Universal Robots PolyScope program: 2024.urp

Program 2024 (installation=default directory=/programs createdIn=5.11.9.1010452 lastSavedIn=5.11.9.1010452 robotSerialNumber=20225200364)
Calibrated DH parameters: a=[0.00002, -0.569483, -0.54992, -0.00001, -0.000036, 0]; d=[0.180894, -146.691669, 192.918669, -46.053088, 0.119778, 0.115602]; alpha=[1.571425, -0.001534, 0.003359, 1.568739, -1.571477, 0]; deltaTheta=[0, 0.376258, -0.101074, -0.275185, -0.000002, 0]
Robot Program (runOnlyOnce=true)
  Script file /programs/usbdisk/new-robot/2024Dragon_V2.script
    | def Machining1():
    |   # Default parameters:
    |   global speed_ms = 0.3
    |   global speed_rads = 0.75
    |   global accel_mss = 3
    |   global accel_radss = 1.2
    |   global blend_radius_m = 0.001
    | 
    |   # Add subprograms here
    |   # Start of main program
    |   # Program generated by RoboDK v5.6.5 for UR10e on 10/01/2024 16:52:19
    |   # Using nominal kinematics.
    |   blend_radius_m = 0.001
    |   speed_ms = 1.000
    |   # set_reference(p[0.320000, -0.152000, -0.016000, 0.000000, 0.000000, 0.000000])
    |   set_tcp(p[0.000000, 0.000000, 0.252000, 0.000000, 0.000000, 0.000000])
    |   # Show Tool
    |   movej([0.070455, -1.061149, -2.628944, -1.022296, 1.570796, 1.641252],accel_radss,speed_rads,0,blend_radius_m)
    |   movel([0.070455, -1.061149, -2.628944, -1.022296, 1.570796, 1.641252],accel_mss,speed_ms,0,blend_radius_m)
    |   # Splitting Linear movement in 30 (instruction 7: MoveL 3)
    |   movel([0.070455, -1.062891, -2.630322, -1.019175, 1.570796, 1.641252],accel_mss,speed_ms,0,blend_radius_m)
    |   movel([0.070455, -1.064646, -2.631698, -1.016044, 1.570796, 1.641252],accel_mss,speed_ms,0,blend_radius_m)
    |   movel([0.070455, -1.066415, -2.633072, -1.012903, 1.570796, 1.641252],accel_mss,speed_ms,0,blend_radius_m)
    |   movel([0.070455, -1.068196, -2.634443, -1.009750, 1.570796, 1.641252],accel_mss,speed_ms,0,blend_radius_m)
    |   movel([0.070455, -1.069991, -2.635811, -1.006586, 1.570796, 1.641252],accel_mss,speed_ms,0,blend_radius_m)
    |   movel([0.070455, -1.071800, -2.637177, -1.003412, 1.570796, 1.641252],accel_mss,speed_ms,0,blend_radius_m)
    |   movel([0.070455, -1.073622, -2.638541, -1.000227, 1.570796, 1.641252],accel_mss,speed_ms,0,blend_radius_m)
    |   movel([0.070455, -1.075457, -2.639902, -0.997030, 1.570796, 1.641252],accel_mss,speed_ms,0,blend_radius_m)
    |   movel([0.070455, -1.077307, -2.641260, -0.993822, 1.570796, 1.641252],accel_mss,speed_ms,0,blend_radius_m)
    |   movel([0.070455, -1.079170, -2.642616, -0.990603, 1.570796, 1.641252],accel_mss,speed_ms,0,blend_radius_m)
    |   movel([0.070455, -1.081047, -2.643969, -0.987373, 1.570796, 1.641252],accel_mss,speed_ms,0,blend_radius_m)
    |   movel([0.070455, -1.082937, -2.645320, -0.984132, 1.570796, 1.641252],accel_mss,speed_ms,0,blend_radius_m)
    |   movel([0.070455, -1.084842, -2.646667, -0.980879, 1.570796, 1.641252],accel_mss,speed_ms,0,blend_radius_m)
    |   movel([0.070455, -1.086761, -2.648013, -0.977615, 1.570796, 1.641252],accel_mss,speed_ms,0,blend_radius_m)
    |   movel([0.070455, -1.088694, -2.649355, -0.974339, 1.570796, 1.641252],accel_mss,speed_ms,0,blend_radius_m)
    |   movel([0.070455, -1.090642, -2.650695, -0.971052, 1.570796, 1.641252],accel_mss,speed_ms,0,blend_radius_m)
    |   movel([0.070455, -1.092603, -2.652032, -0.967753, 1.570796, 1.641252],accel_mss,speed_ms,0,blend_radius_m)
    |   movel([0.070455, -1.094579, -2.653367, -0.964443, 1.570796, 1.641252],accel_mss,speed_ms,0,blend_radius_m)
    |   movel([0.070455, -1.096570, -2.654698, -0.961121, 1.570796, 1.641252],accel_mss,speed_ms,0,blend_radius_m)
    |   movel([0.070455, -1.098575, -2.656027, -0.957787, 1.570796, 1.641252],accel_mss,speed_ms,0,blend_radius_m)
    |   movel([0.070455, -1.100594, -2.657353, -0.954441, 1.570796, 1.641252],accel_mss,speed_ms,0,blend_radius_m)
    |   movel([0.070455, -1.102629, -2.658677, -0.951083, 1.570796, 1.641252],accel_mss,speed_ms,0,blend_radius_m)
    |   movel([0.070455, -1.104678, -2.659997, -0.947714, 1.570796, 1.641252],accel_mss,speed_ms,0,blend_radius_m)
    |   movel([0.070455, -1.106742, -2.661315, -0.944332, 1.570796, 1.641252],accel_mss,speed_ms,0,blend_radius_m)
    |   movel([0.070455, -1.108821, -2.662630, -0.940938, 1.570796, 1.641252],accel_mss,speed_ms,0,blend_radius_m)
    |   movel([0.070455, -1.110915, -2.663942, -0.937533, 1.570796, 1.641252],accel_mss,speed_ms,0,blend_radius_m)
    |   movel([0.070455, -1.113024, -2.665251, -0.934115, 1.570796, 1.641252],accel_mss,speed_ms,0,blend_radius_m)
    |   movel([0.070455, -1.115148, -2.666557, -0.930684, 1.570796, 1.641252],accel_mss,speed_ms,0,blend_radius_m)
    |   movel([0.070455, -1.117287, -2.667860, -0.927242, 1.570796, 1.641252],accel_mss,speed_ms,0,blend_radius_m)
    |   movel([0.070455, -1.119442, -2.669160, -0.923787, 1.570796, 1.641252],accel_mss,speed_ms,0,blend_radius_m)
    |   movel([0.070455, -1.119442, -2.669160, -0.923787, 1.570796, 1.641252],accel_mss,speed_ms,0,blend_radius_m)
    |   speed_ms = 1.000
    |   movel([0.070455, -1.119442, -2.669160, -0.923787, 1.570796, 1.641252],accel_mss,speed_ms,0,blend_radius_m)
    |   movel([0.070455, -1.119442, -2.669160, -0.923787, 1.570796, 1.641252],accel_mss,speed_ms,0,blend_radius_m)
    |   movel([0.070455, -1.119442, -2.669160, -0.923787, 1.570796, 1.641252],accel_mss,speed_ms,0,blend_radius_m)
    |   speed_ms = 0.005
    |   # Splitting Linear movement in 20 (instruction 14: MoveL 8)
    |   movel([0.070455, -1.117287, -2.667860, -0.927242, 1.570796, 1.641252],accel_mss,speed_ms,0,blend_radius_m)
    |   movel([0.070455, -1.115148, -2.666557, -0.930684, 1.570796, 1.641252],accel_mss,speed_ms,0,blend_radius_m)
    |   movel([0.070455, -1.113024, -2.665251, -0.934115, 1.570796, 1.641252],accel_mss,speed_ms,0,blend_radius_m)
    |   movel([0.070455, -1.110915, -2.663942, -0.937533, 1.570796, 1.641252],accel_mss,speed_ms,0,blend_radius_m)
    |   movel([0.070455, -1.108821, -2.662630, -0.940938, 1.570796, 1.641252],accel_mss,speed_ms,0,blend_radius_m)
    |   movel([0.070455, -1.106742, -2.661315, -0.944332, 1.570796, 1.641252],accel_mss,speed_ms,0,blend_radius_m)
    |   movel([0.070455, -1.104678, -2.659997, -0.947714, 1.570796, 1.641252],accel_mss,speed_ms,0,blend_radius_m)
    |   movel([0.070455, -1.102629, -2.658677, -0.951083, 1.570796, 1.641252],accel_mss,speed_ms,0,blend_radius_m)
    |   movel([0.070455, -1.100594, -2.657353, -0.954441, 1.570796, 1.641252],accel_mss,speed_ms,0,blend_radius_m)
    |   movel([0.070455, -1.098575, -2.656027, -0.957787, 1.570796, 1.641252],accel_mss,speed_ms,0,blend_radius_m)
    |   movel([0.070455, -1.096570, -2.654698, -0.961121, 1.570796, 1.641252],accel_mss,speed_ms,0,blend_radius_m)
    |   movel([0.070455, -1.094579, -2.653367, -0.964443, 1.570796, 1.641252],accel_mss,speed_ms,0,blend_radius_m)
    |   movel([0.070455, -1.092603, -2.652032, -0.967753, 1.570796, 1.641252],accel_mss,speed_ms,0,blend_radius_m)
    |   movel([0.070455, -1.090642, -2.650695, -0.971052, 1.570796, 1.641252],accel_mss,speed_ms,0,blend_radius_m)
    |   movel([0.070455, -1.088694, -2.649355, -0.974339, 1.570796, 1.641252],accel_mss,speed_ms,0,blend_radius_m)
    |   movel([0.070455, -1.086761, -2.648013, -0.977615, 1.570796, 1.641252],accel_mss,speed_ms,0,blend_radius_m)
    |   movel([0.070455, -1.084842, -2.646667, -0.980879, 1.570796, 1.641252],accel_mss,speed_ms,0,blend_radius_m)
    |   movel([0.070455, -1.082937, -2.645320, -0.984132, 1.570796, 1.641252],accel_mss,speed_ms,0,blend_radius_m)
    |   movel([0.070455, -1.081047, -2.643969, -0.987373, 1.570796, 1.641252],accel_mss,speed_ms,0,blend_radius_m)
    |   movel([0.070455, -1.079170, -2.642616, -0.990603, 1.570796, 1.641252],accel_mss,speed_ms,0,blend_radius_m)
    |   speed_ms = 1.000
    |   # Splitting Linear movement in 20 (instruction 16: MoveL 9)
    |   movel([0.070455, -1.081047, -2.643969, -0.987373, 1.570796, 1.641252],accel_mss,speed_ms,0,blend_radius_m)
    |   movel([0.070455, -1.082937, -2.645320, -0.984132, 1.570796, 1.641252],accel_mss,speed_ms,0,blend_radius_m)
    |   movel([0.070455, -1.084842, -2.646667, -0.980879, 1.570796, 1.641252],accel_mss,speed_ms,0,blend_radius_m)
    |   movel([0.070455, -1.086761, -2.648013, -0.977615, 1.570796, 1.641252],accel_mss,speed_ms,0,blend_radius_m)
    |   movel([0.070455, -1.088694, -2.649355, -0.974339, 1.570796, 1.641252],accel_mss,speed_ms,0,blend_radius_m)
    |   movel([0.070455, -1.090642, -2.650695, -0.971052, 1.570796, 1.641252],accel_mss,speed_ms,0,blend_radius_m)
    |   movel([0.070455, -1.092603, -2.652032, -0.967753, 1.570796, 1.641252],accel_mss,speed_ms,0,blend_radius_m)
    |   movel([0.070455, -1.094579, -2.653367, -0.964443, 1.570796, 1.641252],accel_mss,speed_ms,0,blend_radius_m)
    |   movel([0.070455, -1.096570, -2.654698, -0.961121, 1.570796, 1.641252],accel_mss,speed_ms,0,blend_radius_m)
    |   movel([0.070455, -1.098575, -2.656027, -0.957787, 1.570796, 1.641252],accel_mss,speed_ms,0,blend_radius_m)
    |   movel([0.070455, -1.100594, -2.657353, -0.954441, 1.570796, 1.641252],accel_mss,speed_ms,0,blend_radius_m)
    |   movel([0.070455, -1.102629, -2.658677, -0.951083, 1.570796, 1.641252],accel_mss,speed_ms,0,blend_radius_m)
    |   movel([0.070455, -1.104678, -2.659997, -0.947714, 1.570796, 1.641252],accel_mss,speed_ms,0,blend_radius_m)
    |   movel([0.070455, -1.106742, -2.661315, -0.944332, 1.570796, 1.641252],accel_mss,speed_ms,0,blend_radius_m)
    |   movel([0.070455, -1.108821, -2.662630, -0.940938, 1.570796, 1.641252],accel_mss,speed_ms,0,blend_radius_m)
    |   movel([0.070455, -1.110915, -2.663942, -0.937533, 1.570796, 1.641252],accel_mss,speed_ms,0,blend_radius_m)
    |   movel([0.070455, -1.113024, -2.665251, -0.934115, 1.570796, 1.641252],accel_mss,speed_ms,0,blend_radius_m)
    |   movel([0.070455, -1.115148, -2.666557, -0.930684, 1.570796, 1.641252],accel_mss,speed_ms,0,blend_radius_m)
    |   movel([0.070455, -1.117287, -2.667860, -0.927242, 1.570796, 1.641252],accel_mss,speed_ms,0,blend_radius_m)
    |   movel([0.070455, -1.119442, -2.669160, -0.923787, 1.570796, 1.641252],accel_mss,speed_ms,0,blend_radius_m)
    |   speed_ms = 0.040
    |   movel([0.070455, -1.119442, -2.669160, -0.923787, 1.570796, 1.641252],accel_mss,speed_ms,0,blend_radius_m)
    |   speed_ms = 1.000
    |   movel([0.070455, -1.119442, -2.669160, -0.923787, 1.570796, 1.641252],accel_mss,speed_ms,0,blend_radius_m)
    |   # Splitting Linear movement in 152 (instruction 21: MoveL 12)
    |   movel([0.070832, -1.122077, -2.668067, -0.922246, 1.570796, 1.641628],accel_mss,speed_ms,0,blend_radius_m)
    |   movel([0.071206, -1.124704, -2.666969, -0.920715, 1.570796, 1.642002],accel_mss,speed_ms,0,blend_radius_m)
    |   movel([0.071578, -1.127324, -2.665869, -0.919196, 1.570796, 1.642374],accel_mss,speed_ms,0,blend_radius_m)
    |   movel([0.071947, -1.129937, -2.664764, -0.917688, 1.570796, 1.642743],accel_mss,speed_ms,0,blend_radius_m)
    |   movel([0.072314, -1.132542, -2.663657, -0.916190, 1.570796, 1.643111],accel_mss,speed_ms,0,blend_radius_m)
    |   movel([0.072679, -1.135140, -2.662545, -0.914703, 1.570796, 1.643476],accel_mss,speed_ms,0,blend_radius_m)
    |   movel([0.073042, -1.137731, -2.661431, -0.913227, 1.570796, 1.643839],accel_mss,speed_ms,0,blend_radius_m)
    |   movel([0.073403, -1.140315, -2.660313, -0.911762, 1.570796, 1.644199],accel_mss,speed_ms,0,blend_radius_m)
    |   movel([0.073761, -1.142891, -2.659192, -0.910307, 1.570796, 1.644558],accel_mss,speed_ms,0,blend_radius_m)
    |   movel([0.074117, -1.145460, -2.658067, -0.908863, 1.570796, 1.644914],accel_mss,speed_ms,0,blend_radius_m)
    |   movel([0.074472, -1.148021, -2.656939, -0.907429, 1.570796, 1.645268],accel_mss,speed_ms,0,blend_radius_m)
    |   movel([0.074824, -1.150576, -2.655807, -0.906006, 1.570796, 1.645620],accel_mss,speed_ms,0,blend_radius_m)
    |   movel([0.075173, -1.153123, -2.654672, -0.904594, 1.570796, 1.645970],accel_mss,speed_ms,0,blend_radius_m)
    |   movel([0.075521, -1.155663, -2.653534, -0.903192, 1.570796, 1.646318],accel_mss,speed_ms,0,blend_radius_m)
    |   movel([0.075867, -1.158196, -2.652393, -0.901800, 1.570796, 1.646663],accel_mss,speed_ms,0,blend_radius_m)
    |   movel([0.076211, -1.160722, -2.651248, -0.900419, 1.570796, 1.647007],accel_mss,speed_ms,0,blend_radius_m)
    |   movel([0.076552, -1.163240, -2.650100, -0.899048, 1.570796, 1.647349],accel_mss,speed_ms,0,blend_radius_m)
    |   movel([0.076892, -1.165752, -2.648949, -0.897688, 1.570796, 1.647688],accel_mss,speed_ms,0,blend_radius_m)
    |   movel([0.077230, -1.168256, -2.647795, -0.896338, 1.570796, 1.648026],accel_mss,speed_ms,0,blend_radius_m)
    |   movel([0.077565, -1.170754, -2.646637, -0.894998, 1.570796, 1.648362],accel_mss,speed_ms,0,blend_radius_m)
    |   movel([0.077899, -1.173244, -2.645477, -0.893668, 1.570796, 1.648695],accel_mss,speed_ms,0,blend_radius_m)
    |   movel([0.078231, -1.175728, -2.644313, -0.892348, 1.570796, 1.649027],accel_mss,speed_ms,0,blend_radius_m)
    |   movel([0.078561, -1.178204, -2.643146, -0.891039, 1.570796, 1.649357],accel_mss,speed_ms,0,blend_radius_m)
    |   movel([0.078888, -1.180674, -2.641976, -0.889739, 1.570796, 1.649685],accel_mss,speed_ms,0,blend_radius_m)
    |   movel([0.079214, -1.183137, -2.640802, -0.888450, 1.570796, 1.650011],accel_mss,speed_ms,0,blend_radius_m)
    |   movel([0.079539, -1.185593, -2.639626, -0.887171, 1.570796, 1.650335],accel_mss,speed_ms,0,blend_radius_m)
    |   movel([0.079861, -1.188042, -2.638446, -0.885901, 1.570796, 1.650657],accel_mss,speed_ms,0,blend_radius_m)
    |   movel([0.080181, -1.190484, -2.637264, -0.884642, 1.570796, 1.650978],accel_mss,speed_ms,0,blend_radius_m)
    |   movel([0.080500, -1.192919, -2.636078, -0.883392, 1.570796, 1.651296],accel_mss,speed_ms,0,blend_radius_m)
    |   movel([0.080817, -1.195347, -2.634889, -0.882152, 1.570796, 1.651613],accel_mss,speed_ms,0,blend_radius_m)
    |   movel([0.081131, -1.197769, -2.633698, -0.880922, 1.570796, 1.651928],accel_mss,speed_ms,0,blend_radius_m)
    |   movel([0.081445, -1.200184, -2.632503, -0.879702, 1.570796, 1.652241],accel_mss,speed_ms,0,blend_radius_m)
    |   movel([0.081756, -1.202593, -2.631305, -0.878491, 1.570796, 1.652552],accel_mss,speed_ms,0,blend_radius_m)
    |   movel([0.082066, -1.204994, -2.630105, -0.877290, 1.570796, 1.652862],accel_mss,speed_ms,0,blend_radius_m)
    |   movel([0.082374, -1.207389, -2.628901, -0.876099, 1.570796, 1.653170],accel_mss,speed_ms,0,blend_radius_m)
    |   movel([0.082680, -1.209777, -2.627694, -0.874917, 1.570796, 1.653476],accel_mss,speed_ms,0,blend_radius_m)
    |   movel([0.082984, -1.212159, -2.626485, -0.873745, 1.570796, 1.653780],accel_mss,speed_ms,0,blend_radius_m)
    |   movel([0.083287, -1.214534, -2.625272, -0.872582, 1.570796, 1.654083],accel_mss,speed_ms,0,blend_radius_m)
    |   movel([0.083588, -1.216903, -2.624057, -0.871429, 1.570796, 1.654384],accel_mss,speed_ms,0,blend_radius_m)
    |   movel([0.083887, -1.219265, -2.622839, -0.870285, 1.570796, 1.654684],accel_mss,speed_ms,0,blend_radius_m)
    |   movel([0.084185, -1.221621, -2.621618, -0.869151, 1.570796, 1.654981],accel_mss,speed_ms,0,blend_radius_m)
    |   movel([0.084481, -1.223970, -2.620394, -0.868026, 1.570796, 1.655277],accel_mss,speed_ms,0,blend_radius_m)
    |   movel([0.084775, -1.226312, -2.619167, -0.866910, 1.570796, 1.655572],accel_mss,speed_ms,0,blend_radius_m)
    |   movel([0.085068, -1.228649, -2.617937, -0.865803, 1.570796, 1.655864],accel_mss,speed_ms,0,blend_radius_m)
    |   movel([0.085359, -1.230978, -2.616705, -0.864706, 1.570796, 1.656156],accel_mss,speed_ms,0,blend_radius_m)
    |   movel([0.085649, -1.233302, -2.615469, -0.863618, 1.570796, 1.656445],accel_mss,speed_ms,0,blend_radius_m)
    |   movel([0.085937, -1.235619, -2.614231, -0.862539, 1.570796, 1.656733],accel_mss,speed_ms,0,blend_radius_m)
    |   movel([0.086223, -1.237930, -2.612991, -0.861468, 1.570796, 1.657020],accel_mss,speed_ms,0,blend_radius_m)
    |   movel([0.086508, -1.240234, -2.611747, -0.860407, 1.570796, 1.657304],accel_mss,speed_ms,0,blend_radius_m)
    |   movel([0.086791, -1.242533, -2.610501, -0.859355, 1.570796, 1.657588],accel_mss,speed_ms,0,blend_radius_m)
    |   movel([0.087073, -1.244825, -2.609252, -0.858312, 1.570796, 1.657869],accel_mss,speed_ms,0,blend_radius_m)
    |   movel([0.087353, -1.247111, -2.608000, -0.857278, 1.570796, 1.658150],accel_mss,speed_ms,0,blend_radius_m)
    |   movel([0.087632, -1.249390, -2.606746, -0.856253, 1.570796, 1.658428],accel_mss,speed_ms,0,blend_radius_m)
    |   movel([0.087909, -1.251664, -2.605488, -0.855237, 1.570796, 1.658706],accel_mss,speed_ms,0,blend_radius_m)
    |   movel([0.088185, -1.253931, -2.604229, -0.854229, 1.570796, 1.658981],accel_mss,speed_ms,0,blend_radius_m)
    |   movel([0.088459, -1.256193, -2.602966, -0.853230, 1.570796, 1.659256],accel_mss,speed_ms,0,blend_radius_m)
    |   movel([0.088732, -1.258448, -2.601701, -0.852240, 1.570796, 1.659528],accel_mss,speed_ms,0,blend_radius_m)
    |   movel([0.089004, -1.260697, -2.600433, -0.851258, 1.570796, 1.659800],accel_mss,speed_ms,0,blend_radius_m)
    |   movel([0.089273, -1.262941, -2.599163, -0.850285, 1.570796, 1.660070],accel_mss,speed_ms,0,blend_radius_m)
    |   movel([0.089542, -1.265178, -2.597890, -0.849321, 1.570796, 1.660338],accel_mss,speed_ms,0,blend_radius_m)
    |   movel([0.089809, -1.267409, -2.596614, -0.848365, 1.570796, 1.660605],accel_mss,speed_ms,0,blend_radius_m)
    |   movel([0.090075, -1.269635, -2.595336, -0.847418, 1.570796, 1.660871],accel_mss,speed_ms,0,blend_radius_m)
    |   movel([0.090339, -1.271854, -2.594055, -0.846479, 1.570796, 1.661135],accel_mss,speed_ms,0,blend_radius_m)
    |   movel([0.090602, -1.274068, -2.592772, -0.845549, 1.570796, 1.661398],accel_mss,speed_ms,0,blend_radius_m)
    |   movel([0.090863, -1.276276, -2.591486, -0.844627, 1.570796, 1.661660],accel_mss,speed_ms,0,blend_radius_m)
    |   movel([0.091123, -1.278478, -2.590198, -0.843713, 1.570796, 1.661920],accel_mss,speed_ms,0,blend_radius_m)
    |   movel([0.091382, -1.280674, -2.588907, -0.842808, 1.570796, 1.662178],accel_mss,speed_ms,0,blend_radius_m)
    |   movel([0.091640, -1.282864, -2.587614, -0.841911, 1.570796, 1.662436],accel_mss,speed_ms,0,blend_radius_m)
    |   movel([0.091896, -1.285049, -2.586318, -0.841022, 1.570796, 1.662692],accel_mss,speed_ms,0,blend_radius_m)
    |   movel([0.092150, -1.287228, -2.585019, -0.840141, 1.570796, 1.662947],accel_mss,speed_ms,0,blend_radius_m)
    |   movel([0.092404, -1.289402, -2.583719, -0.839269, 1.570796, 1.663200],accel_mss,speed_ms,0,blend_radius_m)
    |   movel([0.092656, -1.291569, -2.582415, -0.838404, 1.570796, 1.663452],accel_mss,speed_ms,0,blend_radius_m)
    |   movel([0.092907, -1.293731, -2.581110, -0.837548, 1.570796, 1.663703],accel_mss,speed_ms,0,blend_radius_m)
    |   movel([0.093156, -1.295888, -2.579801, -0.836700, 1.570796, 1.663953],accel_mss,speed_ms,0,blend_radius_m)
    |   movel([0.093405, -1.298039, -2.578491, -0.835859, 1.570796, 1.664201],accel_mss,speed_ms,0,blend_radius_m)
    |   movel([0.093652, -1.300184, -2.577178, -0.835027, 1.570796, 1.664448],accel_mss,speed_ms,0,blend_radius_m)
    |   movel([0.093897, -1.302324, -2.575862, -0.834202, 1.570796, 1.664694],accel_mss,speed_ms,0,blend_radius_m)
    |   movel([0.094142, -1.304459, -2.574545, -0.833386, 1.570796, 1.664938],accel_mss,speed_ms,0,blend_radius_m)
    |   movel([0.094385, -1.306588, -2.573224, -0.832577, 1.570796, 1.665182],accel_mss,speed_ms,0,blend_radius_m)
    |   movel([0.094627, -1.308711, -2.571902, -0.831776, 1.570796, 1.665424],accel_mss,speed_ms,0,blend_radius_m)
    |   movel([0.094868, -1.310829, -2.570577, -0.830983, 1.570796, 1.665664],accel_mss,speed_ms,0,blend_radius_m)
    |   movel([0.095108, -1.312942, -2.569250, -0.830197, 1.570796, 1.665904],accel_mss,speed_ms,0,blend_radius_m)
    |   movel([0.095346, -1.315050, -2.567920, -0.829419, 1.570796, 1.666142],accel_mss,speed_ms,0,blend_radius_m)
    |   movel([0.095583, -1.317152, -2.566588, -0.828649, 1.570796, 1.666380],accel_mss,speed_ms,0,blend_radius_m)
    |   movel([0.095819, -1.319249, -2.565254, -0.827886, 1.570796, 1.666616],accel_mss,speed_ms,0,blend_radius_m)
    |   movel([0.096054, -1.321340, -2.563918, -0.827131, 1.570796, 1.666851],accel_mss,speed_ms,0,blend_radius_m)
    |   movel([0.096288, -1.323427, -2.562579, -0.826384, 1.570796, 1.667084],accel_mss,speed_ms,0,blend_radius_m)
    |   movel([0.096520, -1.325508, -2.561238, -0.825643, 1.570796, 1.667317],accel_mss,speed_ms,0,blend_radius_m)
    |   movel([0.096752, -1.327584, -2.559894, -0.824911, 1.570796, 1.667548],accel_mss,speed_ms,0,blend_radius_m)
    |   movel([0.096982, -1.329654, -2.558549, -0.824186, 1.570796, 1.667778],accel_mss,speed_ms,0,blend_radius_m)
    |   movel([0.097211, -1.331720, -2.557201, -0.823468, 1.570796, 1.668007],accel_mss,speed_ms,0,blend_radius_m)
    |   movel([0.097439, -1.333781, -2.555851, -0.822757, 1.570796, 1.668235],accel_mss,speed_ms,0,blend_radius_m)
    |   movel([0.097666, -1.335836, -2.554499, -0.822054, 1.570796, 1.668462],accel_mss,speed_ms,0,blend_radius_m)
    |   movel([0.097892, -1.337887, -2.553144, -0.821358, 1.570796, 1.668688],accel_mss,speed_ms,0,blend_radius_m)
    |   movel([0.098116, -1.339932, -2.551787, -0.820669, 1.570796, 1.668913],accel_mss,speed_ms,0,blend_radius_m)
    |   movel([0.098340, -1.341972, -2.550429, -0.819988, 1.570796, 1.669136],accel_mss,speed_ms,0,blend_radius_m)
    |   movel([0.098562, -1.344008, -2.549067, -0.819314, 1.570796, 1.669359],accel_mss,speed_ms,0,blend_radius_m)
    |   movel([0.098784, -1.346038, -2.547704, -0.818646, 1.570796, 1.669580],accel_mss,speed_ms,0,blend_radius_m)
    |   movel([0.099004, -1.348064, -2.546339, -0.817986, 1.570796, 1.669800],accel_mss,speed_ms,0,blend_radius_m)
    |   movel([0.099223, -1.350085, -2.544971, -0.817333, 1.570796, 1.670020],accel_mss,speed_ms,0,blend_radius_m)
    |   movel([0.099441, -1.352100, -2.543601, -0.816687, 1.570796, 1.670238],accel_mss,speed_ms,0,blend_radius_m)
    |   movel([0.099659, -1.354111, -2.542230, -0.816048, 1.570796, 1.670455],accel_mss,speed_ms,0,blend_radius_m)
    |   movel([0.099875, -1.356118, -2.540856, -0.815416, 1.570796, 1.670671],accel_mss,speed_ms,0,blend_radius_m)
    |   movel([0.100090, -1.358119, -2.539479, -0.814791, 1.570796, 1.670886],accel_mss,speed_ms,0,blend_radius_m)
    |   movel([0.100304, -1.360116, -2.538101, -0.814172, 1.570796, 1.671100],accel_mss,speed_ms,0,blend_radius_m)
    |   movel([0.100517, -1.362107, -2.536721, -0.813561, 1.570796, 1.671313],accel_mss,speed_ms,0,blend_radius_m)
    |   movel([0.100729, -1.364095, -2.535338, -0.812956, 1.570796, 1.671525],accel_mss,speed_ms,0,blend_radius_m)
    |   movel([0.100940, -1.366077, -2.533954, -0.812358, 1.570796, 1.671736],accel_mss,speed_ms,0,blend_radius_m)
    |   movel([0.101150, -1.368055, -2.532567, -0.811767, 1.570796, 1.671946],accel_mss,speed_ms,0,blend_radius_m)
    |   movel([0.101359, -1.370028, -2.531179, -0.811182, 1.570796, 1.672155],accel_mss,speed_ms,0,blend_radius_m)
    |   movel([0.101567, -1.371997, -2.529788, -0.810604, 1.570796, 1.672363],accel_mss,speed_ms,0,blend_radius_m)
    |   movel([0.101774, -1.373961, -2.528395, -0.810033, 1.570796, 1.672570],accel_mss,speed_ms,0,blend_radius_m)
    |   movel([0.101980, -1.375920, -2.527000, -0.809468, 1.570796, 1.672776],accel_mss,speed_ms,0,blend_radius_m)
    |   movel([0.102185, -1.377875, -2.525604, -0.808910, 1.570796, 1.672981],accel_mss,speed_ms,0,blend_radius_m)
    |   movel([0.102389, -1.379825, -2.524205, -0.808359, 1.570796, 1.673186],accel_mss,speed_ms,0,blend_radius_m)
    |   movel([0.102593, -1.381771, -2.522804, -0.807814, 1.570796, 1.673389],accel_mss,speed_ms,0,blend_radius_m)
    |   movel([0.102795, -1.383713, -2.521401, -0.807275, 1.570796, 1.673591],accel_mss,speed_ms,0,blend_radius_m)
    |   movel([0.102996, -1.385650, -2.519996, -0.806743, 1.570796, 1.673792],accel_mss,speed_ms,0,blend_radius_m)
    |   movel([0.103197, -1.387582, -2.518589, -0.806217, 1.570796, 1.673993],accel_mss,speed_ms,0,blend_radius_m)
    |   movel([0.103396, -1.389510, -2.517181, -0.805698, 1.570796, 1.674192],accel_mss,speed_ms,0,blend_radius_m)
    |   movel([0.103595, -1.391434, -2.515770, -0.805185, 1.570796, 1.674391],accel_mss,speed_ms,0,blend_radius_m)
    |   movel([0.103792, -1.393354, -2.514357, -0.804678, 1.570796, 1.674588],accel_mss,speed_ms,0,blend_radius_m)
    |   movel([0.103989, -1.395269, -2.512942, -0.804178, 1.570796, 1.674785],accel_mss,speed_ms,0,blend_radius_m)
    |   movel([0.104185, -1.397180, -2.511526, -0.803684, 1.570796, 1.674981],accel_mss,speed_ms,0,blend_radius_m)
    |   movel([0.104380, -1.399086, -2.510107, -0.803196, 1.570796, 1.675176],accel_mss,speed_ms,0,blend_radius_m)
    |   movel([0.104574, -1.400989, -2.508686, -0.802714, 1.570796, 1.675370],accel_mss,speed_ms,0,blend_radius_m)
    |   movel([0.104767, -1.402887, -2.507264, -0.802238, 1.570796, 1.675563],accel_mss,speed_ms,0,blend_radius_m)
    |   movel([0.104959, -1.404781, -2.505840, -0.801769, 1.570796, 1.675755],accel_mss,speed_ms,0,blend_radius_m)
    |   movel([0.105151, -1.406670, -2.504413, -0.801305, 1.570796, 1.675947],accel_mss,speed_ms,0,blend_radius_m)
    |   movel([0.105341, -1.408556, -2.502985, -0.800848, 1.570796, 1.676137],accel_mss,speed_ms,0,blend_radius_m)
    |   movel([0.105531, -1.410437, -2.501555, -0.800397, 1.570796, 1.676327],accel_mss,speed_ms,0,blend_radius_m)
    |   movel([0.105720, -1.412315, -2.500123, -0.799951, 1.570796, 1.676516],accel_mss,speed_ms,0,blend_radius_m)
    |   movel([0.105908, -1.414188, -2.498689, -0.799512, 1.570796, 1.676704],accel_mss,speed_ms,0,blend_radius_m)
    |   movel([0.106095, -1.416057, -2.497254, -0.799078, 1.570796, 1.676891],accel_mss,speed_ms,0,blend_radius_m)
    |   movel([0.106281, -1.417922, -2.495816, -0.798651, 1.570796, 1.677077],accel_mss,speed_ms,0,blend_radius_m)
    |   movel([0.106466, -1.419783, -2.494377, -0.798229, 1.570796, 1.677263],accel_mss,speed_ms,0,blend_radius_m)
    |   movel([0.106651, -1.421640, -2.492935, -0.797813, 1.570796, 1.677447],accel_mss,speed_ms,0,blend_radius_m)
    |   movel([0.106835, -1.423494, -2.491492, -0.797403, 1.570796, 1.677631],accel_mss,speed_ms,0,blend_radius_m)
    |   movel([0.107018, -1.425343, -2.490047, -0.796999, 1.570796, 1.677814],accel_mss,speed_ms,0,blend_radius_m)
    |   movel([0.107200, -1.427188, -2.488600, -0.796600, 1.570796, 1.677997],accel_mss,speed_ms,0,blend_radius_m)
    |   movel([0.107382, -1.429030, -2.487152, -0.796208, 1.570796, 1.678178],accel_mss,speed_ms,0,blend_radius_m)
    |   movel([0.107562, -1.430867, -2.485701, -0.795821, 1.570796, 1.678359],accel_mss,speed_ms,0,blend_radius_m)
    |   movel([0.107742, -1.432701, -2.484249, -0.795439, 1.570796, 1.678538],accel_mss,speed_ms,0,blend_radius_m)
    |   movel([0.107921, -1.434531, -2.482795, -0.795063, 1.570796, 1.678717],accel_mss,speed_ms,0,blend_radius_m)
    |   movel([0.108099, -1.436357, -2.481339, -0.794693, 1.570796, 1.678896],accel_mss,speed_ms,0,blend_radius_m)
    |   movel([0.108277, -1.438179, -2.479881, -0.794329, 1.570796, 1.679073],accel_mss,speed_ms,0,blend_radius_m)
    |   movel([0.108453, -1.439997, -2.478422, -0.793970, 1.570796, 1.679250],accel_mss,speed_ms,0,blend_radius_m)
    |   movel([0.108629, -1.441812, -2.476961, -0.793616, 1.570796, 1.679426],accel_mss,speed_ms,0,blend_radius_m)
    |   movel([0.108804, -1.443623, -2.475498, -0.793268, 1.570796, 1.679601],accel_mss,speed_ms,0,blend_radius_m)
    |   movel([0.108979, -1.445430, -2.474033, -0.792926, 1.570796, 1.679775],accel_mss,speed_ms,0,blend_radius_m)
    |   movel([0.109152, -1.447233, -2.472567, -0.792589, 1.570796, 1.679949],accel_mss,speed_ms,0,blend_radius_m)
    |   movel([0.109325, -1.449033, -2.471098, -0.792257, 1.570796, 1.680122],accel_mss,speed_ms,0,blend_radius_m)
    |   speed_ms = 0.005
    |   # Splitting Linear movement in 20 (instruction 23: MoveL 13)
    |   movel([0.109325, -1.450882, -2.472048, -0.789459, 1.570796, 1.680122],accel_mss,speed_ms,0,blend_radius_m)
    |   movel([0.109325, -1.452738, -2.472994, -0.786657, 1.570796, 1.680122],accel_mss,speed_ms,0,blend_radius_m)
    |   movel([0.109325, -1.454601, -2.473936, -0.783852, 1.570796, 1.680122],accel_mss,speed_ms,0,blend_radius_m)
    |   movel([0.109325, -1.456472, -2.474875, -0.781042, 1.570796, 1.680122],accel_mss,speed_ms,0,blend_radius_m)
    |   movel([0.109325, -1.458351, -2.475811, -0.778228, 1.570796, 1.680122],accel_mss,speed_ms,0,blend_radius_m)
    |   movel([0.109325, -1.460236, -2.476742, -0.775410, 1.570796, 1.680122],accel_mss,speed_ms,0,blend_radius_m)
    |   movel([0.109325, -1.462130, -2.477671, -0.772588, 1.570796, 1.680122],accel_mss,speed_ms,0,blend_radius_m)
    |   movel([0.109325, -1.464030, -2.478596, -0.769763, 1.570796, 1.680122],accel_mss,speed_ms,0,blend_radius_m)
    |   movel([0.109325, -1.465939, -2.479517, -0.766933, 1.570796, 1.680122],accel_mss,speed_ms,0,blend_radius_m)
    |   movel([0.109325, -1.467854, -2.480435, -0.764100, 1.570796, 1.680122],accel_mss,speed_ms,0,blend_radius_m)
    |   movel([0.109325, -1.469778, -2.481349, -0.761262, 1.570796, 1.680122],accel_mss,speed_ms,0,blend_radius_m)
    |   movel([0.109325, -1.471708, -2.482260, -0.758421, 1.570796, 1.680122],accel_mss,speed_ms,0,blend_radius_m)
    |   movel([0.109325, -1.473646, -2.483166, -0.755576, 1.570796, 1.680122],accel_mss,speed_ms,0,blend_radius_m)
    |   movel([0.109325, -1.475592, -2.484070, -0.752727, 1.570796, 1.680122],accel_mss,speed_ms,0,blend_radius_m)
    |   movel([0.109325, -1.477545, -2.484970, -0.749874, 1.570796, 1.680122],accel_mss,speed_ms,0,blend_radius_m)
    |   movel([0.109325, -1.479506, -2.485866, -0.747018, 1.570796, 1.680122],accel_mss,speed_ms,0,blend_radius_m)
    |   movel([0.109325, -1.481474, -2.486758, -0.744157, 1.570796, 1.680122],accel_mss,speed_ms,0,blend_radius_m)
    |   movel([0.109325, -1.483449, -2.487647, -0.741293, 1.570796, 1.680122],accel_mss,speed_ms,0,blend_radius_m)
    |   movel([0.109325, -1.485432, -2.488532, -0.738425, 1.570796, 1.680122],accel_mss,speed_ms,0,blend_radius_m)
    |   movel([0.109325, -1.487423, -2.489414, -0.735553, 1.570796, 1.680122],accel_mss,speed_ms,0,blend_radius_m)
    |   speed_ms = 0.035
    |   movel([0.106390, -1.488332, -2.488625, -0.735432, 1.570796, 1.677187],accel_mss,speed_ms,0,blend_radius_m)
    |   movel([0.104973, -1.488645, -2.488353, -0.735391, 1.570796, 1.675769],accel_mss,speed_ms,0,blend_radius_m)
    |   movel([0.103601, -1.488832, -2.488191, -0.735367, 1.570796, 1.674397],accel_mss,speed_ms,0,blend_radius_m)
    |   movel([0.102288, -1.488872, -2.488155, -0.735361, 1.570796, 1.673084],accel_mss,speed_ms,0,blend_radius_m)
    |   movel([0.101045, -1.488742, -2.488269, -0.735378, 1.570796, 1.671842],accel_mss,speed_ms,0,blend_radius_m)
    |   movel([0.099883, -1.488417, -2.488551, -0.735421, 1.570796, 1.670680],accel_mss,speed_ms,0,blend_radius_m)
    |   movel([0.098812, -1.487874, -2.489022, -0.735493, 1.570796, 1.669608],accel_mss,speed_ms,0,blend_radius_m)
    |   movel([0.097838, -1.487097, -2.489696, -0.735596, 1.570796, 1.668635],accel_mss,speed_ms,0,blend_radius_m)
    |   movel([0.097119, -1.486197, -2.490475, -0.735717, 1.570796, 1.667915],accel_mss,speed_ms,0,blend_radius_m)
    |   movel([0.096647, -1.485185, -2.491349, -0.735854, 1.570796, 1.667444],accel_mss,speed_ms,0,blend_radius_m)
    |   movel([0.096406, -1.484067, -2.492314, -0.736008, 1.570796, 1.667202],accel_mss,speed_ms,0,blend_radius_m)
    |   movel([0.096389, -1.482855, -2.493357, -0.736177, 1.570796, 1.667185],accel_mss,speed_ms,0,blend_radius_m)
    |   movel([0.096585, -1.481557, -2.494472, -0.736360, 1.570796, 1.667381],accel_mss,speed_ms,0,blend_radius_m)
    |   movel([0.096979, -1.480185, -2.495647, -0.736557, 1.570796, 1.667776],accel_mss,speed_ms,0,blend_radius_m)
    |   movel([0.097567, -1.478744, -2.496878, -0.736767, 1.570796, 1.668363],accel_mss,speed_ms,0,blend_radius_m)
    |   movel([0.098140, -1.477622, -2.497835, -0.736932, 1.570796, 1.668937],accel_mss,speed_ms,0,blend_radius_m)
    |   movel([0.098807, -1.476536, -2.498759, -0.737094, 1.570796, 1.669603],accel_mss,speed_ms,0,blend_radius_m)
    |   movel([0.099565, -1.475487, -2.499650, -0.737253, 1.570796, 1.670362],accel_mss,speed_ms,0,blend_radius_m)
    |   movel([0.100412, -1.474478, -2.500504, -0.737407, 1.570796, 1.671208],accel_mss,speed_ms,0,blend_radius_m)
    |   movel([0.101347, -1.473511, -2.501322, -0.737556, 1.570796, 1.672143],accel_mss,speed_ms,0,blend_radius_m)
    |   movel([0.102367, -1.472587, -2.502102, -0.737699, 1.570796, 1.673163],accel_mss,speed_ms,0,blend_radius_m)
    |   movel([0.103473, -1.471710, -2.502842, -0.737837, 1.570796, 1.674269],accel_mss,speed_ms,0,blend_radius_m)
    |   movel([0.107265, -1.469032, -2.505092, -0.738265, 1.570796, 1.678061],accel_mss,speed_ms,0,blend_radius_m)
    |   movel([0.109584, -1.467092, -2.506715, -0.738582, 1.570796, 1.680380],accel_mss,speed_ms,0,blend_radius_m)
    |   movel([0.111609, -1.465058, -2.508410, -0.738920, 1.570796, 1.682406],accel_mss,speed_ms,0,blend_radius_m)
    |   movel([0.113340, -1.462927, -2.510180, -0.739282, 1.570796, 1.684137],accel_mss,speed_ms,0,blend_radius_m)
    |   movel([0.114773, -1.460697, -2.512024, -0.739668, 1.570796, 1.685569],accel_mss,speed_ms,0,blend_radius_m)
    |   movel([0.115901, -1.458366, -2.513944, -0.740080, 1.570796, 1.686697],accel_mss,speed_ms,0,blend_radius_m)
    |   movel([0.116721, -1.455930, -2.515940, -0.740519, 1.570796, 1.687517],accel_mss,speed_ms,0,blend_radius_m)
    |   movel([0.117230, -1.453392, -2.518011, -0.740986, 1.570796, 1.688027],accel_mss,speed_ms,0,blend_radius_m)
    |   movel([0.117388, -1.452713, -2.518564, -0.741113, 1.570796, 1.688184],accel_mss,speed_ms,0,blend_radius_m)
    |   movel([0.117692, -1.452199, -2.518981, -0.741209, 1.570796, 1.688488],accel_mss,speed_ms,0,blend_radius_m)
    |   movel([0.118214, -1.451822, -2.519287, -0.741280, 1.570796, 1.689011],accel_mss,speed_ms,0,blend_radius_m)
    |   movel([0.119019, -1.451560, -2.519500, -0.741330, 1.570796, 1.689815],accel_mss,speed_ms,0,blend_radius_m)
    |   movel([0.119828, -1.451443, -2.519594, -0.741352, 1.570796, 1.690624],accel_mss,speed_ms,0,blend_radius_m)
    |   movel([0.120369, -1.451543, -2.519513, -0.741333, 1.570796, 1.691165],accel_mss,speed_ms,0,blend_radius_m)
    |   movel([0.120635, -1.451922, -2.519206, -0.741261, 1.570796, 1.691431],accel_mss,speed_ms,0,blend_radius_m)
    |   movel([0.120635, -1.452630, -2.518631, -0.741128, 1.570796, 1.691431],accel_mss,speed_ms,0,blend_radius_m)
    |   movel([0.120005, -1.455545, -2.516255, -0.740589, 1.570796, 1.690801],accel_mss,speed_ms,0,blend_radius_m)
    |   movel([0.119559, -1.456959, -2.515098, -0.740332, 1.570796, 1.690356],accel_mss,speed_ms,0,blend_radius_m)
    |   movel([0.118418, -1.459695, -2.512850, -0.739844, 1.570796, 1.689214],accel_mss,speed_ms,0,blend_radius_m)
    |   movel([0.117722, -1.461020, -2.511758, -0.739612, 1.570796, 1.688518],accel_mss,speed_ms,0,blend_radius_m)
    |   movel([0.116082, -1.463586, -2.509634, -0.739169, 1.570796, 1.686878],accel_mss,speed_ms,0,blend_radius_m)
    |   movel([0.115138, -1.464828, -2.508602, -0.738959, 1.570796, 1.685935],accel_mss,speed_ms,0,blend_radius_m)
    |   movel([0.113008, -1.467235, -2.506595, -0.738558, 1.570796, 1.683804],accel_mss,speed_ms,0,blend_radius_m)
    |   movel([0.111821, -1.468403, -2.505619, -0.738367, 1.570796, 1.682617],accel_mss,speed_ms,0,blend_radius_m)
    |   movel([0.109208, -1.470664, -2.503722, -0.738003, 1.570796, 1.680005],accel_mss,speed_ms,0,blend_radius_m)
    |   movel([0.106281, -1.472834, -2.501894, -0.737661, 1.570796, 1.677078],accel_mss,speed_ms,0,blend_radius_m)
    |   movel([0.104993, -1.473809, -2.501071, -0.737510, 1.570796, 1.675790],accel_mss,speed_ms,0,blend_radius_m)
    |   movel([0.103770, -1.474892, -2.500153, -0.737343, 1.570796, 1.674567],accel_mss,speed_ms,0,blend_radius_m)
    |   movel([0.102637, -1.476047, -2.499174, -0.737168, 1.570796, 1.673433],accel_mss,speed_ms,0,blend_radius_m)
    |   movel([0.101614, -1.477232, -2.498166, -0.736990, 1.570796, 1.672410],accel_mss,speed_ms,0,blend_radius_m)
    |   movel([0.100892, -1.478221, -2.497324, -0.736844, 1.570796, 1.671688],accel_mss,speed_ms,0,blend_radius_m)
    |   movel([0.100333, -1.479195, -2.496493, -0.736701, 1.570796, 1.671129],accel_mss,speed_ms,0,blend_radius_m)
    |   movel([0.099937, -1.480149, -2.495678, -0.736562, 1.570796, 1.670734],accel_mss,speed_ms,0,blend_radius_m)
    |   movel([0.099701, -1.481076, -2.494884, -0.736429, 1.570796, 1.670497],accel_mss,speed_ms,0,blend_radius_m)
    |   movel([0.099625, -1.481975, -2.494113, -0.736301, 1.570796, 1.670421],accel_mss,speed_ms,0,blend_radius_m)
    |   movel([0.099708, -1.482839, -2.493371, -0.736179, 1.570796, 1.670504],accel_mss,speed_ms,0,blend_radius_m)
    |   movel([0.099948, -1.483663, -2.492662, -0.736064, 1.570796, 1.670745],accel_mss,speed_ms,0,blend_radius_m)
    |   movel([0.100345, -1.484445, -2.491988, -0.735956, 1.570796, 1.671142],accel_mss,speed_ms,0,blend_radius_m)
    |   movel([0.100864, -1.485081, -2.491439, -0.735869, 1.570796, 1.671661],accel_mss,speed_ms,0,blend_radius_m)
    |   movel([0.101501, -1.485533, -2.491049, -0.735807, 1.570796, 1.672297],accel_mss,speed_ms,0,blend_radius_m)
    |   movel([0.102239, -1.485826, -2.490796, -0.735767, 1.570796, 1.673035],accel_mss,speed_ms,0,blend_radius_m)
    |   movel([0.103062, -1.485978, -2.490665, -0.735747, 1.570796, 1.673859],accel_mss,speed_ms,0,blend_radius_m)
    |   movel([0.103963, -1.486005, -2.490641, -0.735743, 1.570796, 1.674759],accel_mss,speed_ms,0,blend_radius_m)
    |   movel([0.104925, -1.485928, -2.490708, -0.735753, 1.570796, 1.675721],accel_mss,speed_ms,0,blend_radius_m)
    |   movel([0.108488, -1.485221, -2.491319, -0.735849, 1.570796, 1.679285],accel_mss,speed_ms,0,blend_radius_m)
    |   movel([0.108948, -1.485204, -2.491333, -0.735852, 1.570796, 1.679745],accel_mss,speed_ms,0,blend_radius_m)
    |   movel([0.109247, -1.485313, -2.491239, -0.735837, 1.570796, 1.680043],accel_mss,speed_ms,0,blend_radius_m)
    |   movel([0.109406, -1.485569, -2.491018, -0.735802, 1.570796, 1.680203],accel_mss,speed_ms,0,blend_radius_m)
    |   movel([0.109457, -1.485990, -2.490654, -0.735745, 1.570796, 1.680253],accel_mss,speed_ms,0,blend_radius_m)
    |   movel([0.109325, -1.487423, -2.489414, -0.735553, 1.570796, 1.680122],accel_mss,speed_ms,0,blend_radius_m)
    |   movel([0.107114, -1.488106, -2.488821, -0.735462, 1.570796, 1.677911],accel_mss,speed_ms,0,blend_radius_m)
    |   speed_ms = 0.005
    |   # Splitting Linear movement in 6 (instruction 99: MoveL 87)
    |   movel([0.107114, -1.486779, -2.488234, -0.737376, 1.570796, 1.677911],accel_mss,speed_ms,0,blend_radius_m)
    |   movel([0.107114, -1.485456, -2.487645, -0.739288, 1.570796, 1.677911],accel_mss,speed_ms,0,blend_radius_m)
    |   movel([0.107114, -1.484136, -2.487055, -0.741198, 1.570796, 1.677911],accel_mss,speed_ms,0,blend_radius_m)
    |   movel([0.107114, -1.482819, -2.486464, -0.743107, 1.570796, 1.677911],accel_mss,speed_ms,0,blend_radius_m)
    |   movel([0.107114, -1.481505, -2.485870, -0.745014, 1.570796, 1.677911],accel_mss,speed_ms,0,blend_radius_m)
    |   movel([0.107114, -1.480195, -2.485275, -0.746919, 1.570796, 1.677911],accel_mss,speed_ms,0,blend_radius_m)
    |   speed_ms = 0.040
    |   # Splitting Linear movement in 14 (instruction 101: MoveL 88)
    |   movel([0.106275, -1.478838, -2.486437, -0.747114, 1.570796, 1.677072],accel_mss,speed_ms,0,blend_radius_m)
    |   movel([0.105433, -1.477481, -2.487596, -0.747312, 1.570796, 1.676230],accel_mss,speed_ms,0,blend_radius_m)
    |   movel([0.104588, -1.476124, -2.488752, -0.747513, 1.570796, 1.675384],accel_mss,speed_ms,0,blend_radius_m)
    |   movel([0.103740, -1.474765, -2.489907, -0.747717, 1.570796, 1.674536],accel_mss,speed_ms,0,blend_radius_m)
    |   movel([0.102889, -1.473406, -2.491059, -0.747924, 1.570796, 1.673685],accel_mss,speed_ms,0,blend_radius_m)
    |   movel([0.102034, -1.472046, -2.492209, -0.748134, 1.570796, 1.672831],accel_mss,speed_ms,0,blend_radius_m)
    |   movel([0.101177, -1.470685, -2.493357, -0.748347, 1.570796, 1.671973],accel_mss,speed_ms,0,blend_radius_m)
    |   movel([0.100316, -1.469323, -2.494503, -0.748563, 1.570796, 1.671112],accel_mss,speed_ms,0,blend_radius_m)
    |   movel([0.099452, -1.467961, -2.495647, -0.748782, 1.570796, 1.670249],accel_mss,speed_ms,0,blend_radius_m)
    |   movel([0.098585, -1.466598, -2.496788, -0.749003, 1.570796, 1.669382],accel_mss,speed_ms,0,blend_radius_m)
    |   movel([0.097715, -1.465234, -2.497927, -0.749228, 1.570796, 1.668512],accel_mss,speed_ms,0,blend_radius_m)
    |   movel([0.096842, -1.463869, -2.499064, -0.749456, 1.570796, 1.667638],accel_mss,speed_ms,0,blend_radius_m)
    |   movel([0.095965, -1.462504, -2.500199, -0.749687, 1.570796, 1.666762],accel_mss,speed_ms,0,blend_radius_m)
    |   movel([0.095086, -1.461137, -2.501331, -0.749921, 1.570796, 1.665882],accel_mss,speed_ms,0,blend_radius_m)
    |   speed_ms = 0.005
    |   # Splitting Linear movement in 4 (instruction 103: MoveL 89)
    |   movel([0.095086, -1.463141, -2.502242, -0.747006, 1.570796, 1.665882],accel_mss,speed_ms,0,blend_radius_m)
    |   movel([0.095086, -1.465152, -2.503149, -0.744088, 1.570796, 1.665882],accel_mss,speed_ms,0,blend_radius_m)
    |   movel([0.095086, -1.467171, -2.504053, -0.741165, 1.570796, 1.665882],accel_mss,speed_ms,0,blend_radius_m)
    |   movel([0.095086, -1.469198, -2.504953, -0.738238, 1.570796, 1.665882],accel_mss,speed_ms,0,blend_radius_m)
    |   speed_ms = 0.035
    |   movel([0.094408, -1.467072, -2.506732, -0.738585, 1.570796, 1.665204],accel_mss,speed_ms,0,blend_radius_m)
    |   movel([0.097635, -1.464926, -2.508520, -0.738943, 1.570796, 1.668431],accel_mss,speed_ms,0,blend_radius_m)
    |   movel([0.098819, -1.464029, -2.509266, -0.739094, 1.570796, 1.669615],accel_mss,speed_ms,0,blend_radius_m)
    |   movel([0.099893, -1.463093, -2.510042, -0.739254, 1.570796, 1.670689],accel_mss,speed_ms,0,blend_radius_m)
    |   movel([0.100845, -1.462120, -2.510848, -0.739421, 1.570796, 1.671641],accel_mss,speed_ms,0,blend_radius_m)
    |   movel([0.101674, -1.461108, -2.511685, -0.739596, 1.570796, 1.672470],accel_mss,speed_ms,0,blend_radius_m)
    |   movel([0.102366, -1.460053, -2.512555, -0.739781, 1.570796, 1.673162],accel_mss,speed_ms,0,blend_radius_m)
    |   movel([0.102914, -1.458956, -2.513459, -0.739975, 1.570796, 1.673710],accel_mss,speed_ms,0,blend_radius_m)
    |   movel([0.103311, -1.457818, -2.514394, -0.740178, 1.570796, 1.674107],accel_mss,speed_ms,0,blend_radius_m)
    |   movel([0.103546, -1.456634, -2.515364, -0.740391, 1.570796, 1.674342],accel_mss,speed_ms,0,blend_radius_m)
    |   movel([0.103749, -1.455882, -2.515980, -0.740528, 1.570796, 1.674545],accel_mss,speed_ms,0,blend_radius_m)
    |   movel([0.104143, -1.455363, -2.516404, -0.740622, 1.570796, 1.674939],accel_mss,speed_ms,0,blend_radius_m)
    |   movel([0.104744, -1.455007, -2.516694, -0.740688, 1.570796, 1.675540],accel_mss,speed_ms,0,blend_radius_m)
    |   movel([0.105564, -1.454746, -2.516907, -0.740735, 1.570796, 1.676361],accel_mss,speed_ms,0,blend_radius_m)
    |   movel([0.106357, -1.454639, -2.516995, -0.740755, 1.570796, 1.677153],accel_mss,speed_ms,0,blend_radius_m)
    |   movel([0.106803, -1.454800, -2.516863, -0.740725, 1.570796, 1.677599],accel_mss,speed_ms,0,blend_radius_m)
    |   movel([0.106975, -1.455210, -2.516529, -0.740650, 1.570796, 1.677772],accel_mss,speed_ms,0,blend_radius_m)
    |   movel([0.106958, -1.455842, -2.516012, -0.740535, 1.570796, 1.677754],accel_mss,speed_ms,0,blend_radius_m)
    |   movel([0.106539, -1.457716, -2.514477, -0.740196, 1.570796, 1.677335],accel_mss,speed_ms,0,blend_radius_m)
    |   movel([0.105755, -1.459606, -2.512924, -0.739860, 1.570796, 1.676551],accel_mss,speed_ms,0,blend_radius_m)
    |   movel([0.104635, -1.461473, -2.511383, -0.739533, 1.570796, 1.675431],accel_mss,speed_ms,0,blend_radius_m)
    |   movel([0.103212, -1.463278, -2.509889, -0.739222, 1.570796, 1.674008],accel_mss,speed_ms,0,blend_radius_m)
    |   movel([0.101515, -1.464990, -2.508467, -0.738932, 1.570796, 1.672311],accel_mss,speed_ms,0,blend_radius_m)
    |   movel([0.099576, -1.466569, -2.507152, -0.738668, 1.570796, 1.670372],accel_mss,speed_ms,0,blend_radius_m)
    |   movel([0.097423, -1.467983, -2.505970, -0.738436, 1.570796, 1.668219],accel_mss,speed_ms,0,blend_radius_m)
    |   movel([0.095086, -1.469198, -2.504953, -0.738238, 1.570796, 1.665882],accel_mss,speed_ms,0,blend_radius_m)
    |   movel([0.094565, -1.467566, -2.506319, -0.738504, 1.570796, 1.665362],accel_mss,speed_ms,0,blend_radius_m)
    |   speed_ms = 0.005
    |   # Splitting Linear movement in 6 (instruction 133: MoveL 117)
    |   movel([0.094565, -1.466211, -2.505719, -0.740459, 1.570796, 1.665362],accel_mss,speed_ms,0,blend_radius_m)
    |   movel([0.094565, -1.464860, -2.505116, -0.742412, 1.570796, 1.665362],accel_mss,speed_ms,0,blend_radius_m)
    |   movel([0.094565, -1.463513, -2.504513, -0.744363, 1.570796, 1.665362],accel_mss,speed_ms,0,blend_radius_m)
    |   movel([0.094565, -1.462169, -2.503907, -0.746313, 1.570796, 1.665362],accel_mss,speed_ms,0,blend_radius_m)
    |   movel([0.094565, -1.460829, -2.503300, -0.748260, 1.570796, 1.665362],accel_mss,speed_ms,0,blend_radius_m)
    |   movel([0.094565, -1.459492, -2.502691, -0.750206, 1.570796, 1.665362],accel_mss,speed_ms,0,blend_radius_m)
    |   speed_ms = 0.040
    |   # Splitting Linear movement in 18 (instruction 135: MoveL 118)
    |   movel([0.094508, -1.457777, -2.504104, -0.750508, 1.570796, 1.665304],accel_mss,speed_ms,0,blend_radius_m)
    |   movel([0.094450, -1.456058, -2.505516, -0.750815, 1.570796, 1.665246],accel_mss,speed_ms,0,blend_radius_m)
    |   movel([0.094391, -1.454335, -2.506927, -0.751127, 1.570796, 1.665188],accel_mss,speed_ms,0,blend_radius_m)
    |   movel([0.094333, -1.452608, -2.508336, -0.751445, 1.570796, 1.665129],accel_mss,speed_ms,0,blend_radius_m)
    |   movel([0.094274, -1.450878, -2.509744, -0.751767, 1.570796, 1.665071],accel_mss,speed_ms,0,blend_radius_m)
    |   movel([0.094215, -1.449143, -2.511150, -0.752095, 1.570796, 1.665012],accel_mss,speed_ms,0,blend_radius_m)
    |   movel([0.094156, -1.447405, -2.512555, -0.752429, 1.570796, 1.664952],accel_mss,speed_ms,0,blend_radius_m)
    |   movel([0.094097, -1.445663, -2.513959, -0.752767, 1.570796, 1.664893],accel_mss,speed_ms,0,blend_radius_m)
    |   movel([0.094037, -1.443917, -2.515361, -0.753112, 1.570796, 1.664833],accel_mss,speed_ms,0,blend_radius_m)
    |   movel([0.093977, -1.442167, -2.516761, -0.753461, 1.570796, 1.664773],accel_mss,speed_ms,0,blend_radius_m)
    |   movel([0.093917, -1.440413, -2.518160, -0.753816, 1.570796, 1.664713],accel_mss,speed_ms,0,blend_radius_m)
    |   movel([0.093856, -1.438655, -2.519558, -0.754176, 1.570796, 1.664653],accel_mss,speed_ms,0,blend_radius_m)
    |   movel([0.093796, -1.436893, -2.520954, -0.754542, 1.570796, 1.664592],accel_mss,speed_ms,0,blend_radius_m)
    |   movel([0.093735, -1.435127, -2.522348, -0.754914, 1.570796, 1.664531],accel_mss,speed_ms,0,blend_radius_m)
    |   movel([0.093673, -1.433357, -2.523741, -0.755291, 1.570796, 1.664470],accel_mss,speed_ms,0,blend_radius_m)
    |   movel([0.093612, -1.431583, -2.525133, -0.755673, 1.570796, 1.664408],accel_mss,speed_ms,0,blend_radius_m)
    |   movel([0.093550, -1.429805, -2.526523, -0.756061, 1.570796, 1.664346],accel_mss,speed_ms,0,blend_radius_m)
    |   movel([0.093488, -1.428022, -2.527912, -0.756455, 1.570796, 1.664284],accel_mss,speed_ms,0,blend_radius_m)
    |   speed_ms = 0.005
    |   # Splitting Linear movement in 6 (instruction 137: MoveL 119)
    |   movel([0.093488, -1.429398, -2.528542, -0.754448, 1.570796, 1.664284],accel_mss,speed_ms,0,blend_radius_m)
    |   movel([0.093488, -1.430779, -2.529171, -0.752440, 1.570796, 1.664284],accel_mss,speed_ms,0,blend_radius_m)
    |   movel([0.093488, -1.432163, -2.529798, -0.750429, 1.570796, 1.664284],accel_mss,speed_ms,0,blend_radius_m)
    |   movel([0.093488, -1.433550, -2.530423, -0.748415, 1.570796, 1.664284],accel_mss,speed_ms,0,blend_radius_m)
    |   movel([0.093488, -1.434942, -2.531047, -0.746400, 1.570796, 1.664284],accel_mss,speed_ms,0,blend_radius_m)
    |   movel([0.093488, -1.436337, -2.531669, -0.744382, 1.570796, 1.664284],accel_mss,speed_ms,0,blend_radius_m)
    |   speed_ms = 0.035
    |   # Splitting Linear movement in 4 (instruction 139: MoveL 120)
    |   movel([0.095293, -1.435866, -2.532041, -0.744482, 1.570796, 1.666089],accel_mss,speed_ms,0,blend_radius_m)
    |   movel([0.097098, -1.435397, -2.532410, -0.744582, 1.570796, 1.667895],accel_mss,speed_ms,0,blend_radius_m)
    |   movel([0.098905, -1.434930, -2.532777, -0.744682, 1.570796, 1.669701],accel_mss,speed_ms,0,blend_radius_m)
    |   movel([0.100712, -1.434465, -2.533142, -0.744782, 1.570796, 1.671508],accel_mss,speed_ms,0,blend_radius_m)
    |   movel([0.101513, -1.434332, -2.533247, -0.744811, 1.570796, 1.672310],accel_mss,speed_ms,0,blend_radius_m)
    |   movel([0.102000, -1.434467, -2.533140, -0.744782, 1.570796, 1.672796],accel_mss,speed_ms,0,blend_radius_m)
    |   movel([0.102216, -1.434868, -2.532826, -0.744696, 1.570796, 1.673012],accel_mss,speed_ms,0,blend_radius_m)
    |   movel([0.102214, -1.435527, -2.532307, -0.744555, 1.570796, 1.673011],accel_mss,speed_ms,0,blend_radius_m)
    |   movel([0.102036, -1.436238, -2.531748, -0.744403, 1.570796, 1.672832],accel_mss,speed_ms,0,blend_radius_m)
    |   movel([0.101677, -1.436767, -2.531331, -0.744291, 1.570796, 1.672474],accel_mss,speed_ms,0,blend_radius_m)
    |   movel([0.101110, -1.437149, -2.531029, -0.744210, 1.570796, 1.671906],accel_mss,speed_ms,0,blend_radius_m)
    |   movel([0.100306, -1.437422, -2.530814, -0.744153, 1.570796, 1.671102],accel_mss,speed_ms,0,blend_radius_m)
    |   # Splitting Linear movement in 8 (instruction 148: MoveL 129)
    |   movel([0.098506, -1.437877, -2.530455, -0.744057, 1.570796, 1.669303],accel_mss,speed_ms,0,blend_radius_m)
    |   movel([0.096708, -1.438333, -2.530094, -0.743962, 1.570796, 1.667504],accel_mss,speed_ms,0,blend_radius_m)
    |   movel([0.094909, -1.438792, -2.529731, -0.743866, 1.570796, 1.665706],accel_mss,speed_ms,0,blend_radius_m)
    |   movel([0.093112, -1.439253, -2.529366, -0.743770, 1.570796, 1.663908],accel_mss,speed_ms,0,blend_radius_m)
    |   movel([0.091315, -1.439716, -2.528999, -0.743674, 1.570796, 1.662111],accel_mss,speed_ms,0,blend_radius_m)
    |   movel([0.089519, -1.440181, -2.528630, -0.743578, 1.570796, 1.660315],accel_mss,speed_ms,0,blend_radius_m)
    |   movel([0.087724, -1.440648, -2.528259, -0.743482, 1.570796, 1.658520],accel_mss,speed_ms,0,blend_radius_m)
    |   movel([0.085929, -1.441117, -2.527886, -0.743386, 1.570796, 1.656725],accel_mss,speed_ms,0,blend_radius_m)
    |   movel([0.085098, -1.441257, -2.527775, -0.743357, 1.570796, 1.655894],accel_mss,speed_ms,0,blend_radius_m)
    |   movel([0.084565, -1.441138, -2.527869, -0.743381, 1.570796, 1.655361],accel_mss,speed_ms,0,blend_radius_m)
    |   movel([0.084301, -1.440737, -2.528189, -0.743464, 1.570796, 1.655097],accel_mss,speed_ms,0,blend_radius_m)
    |   movel([0.084287, -1.440029, -2.528751, -0.743609, 1.570796, 1.655084],accel_mss,speed_ms,0,blend_radius_m)
    |   movel([0.084500, -1.439284, -2.529341, -0.743764, 1.570796, 1.655297],accel_mss,speed_ms,0,blend_radius_m)
    |   movel([0.084917, -1.438781, -2.529739, -0.743868, 1.570796, 1.655713],accel_mss,speed_ms,0,blend_radius_m)
    |   movel([0.085517, -1.438452, -2.530000, -0.743937, 1.570796, 1.656313],accel_mss,speed_ms,0,blend_radius_m)
    |   movel([0.086281, -1.438217, -2.530186, -0.743986, 1.570796, 1.657077],accel_mss,speed_ms,0,blend_radius_m)
    |   # Splitting Linear movement in 4 (instruction 157: MoveL 138)
    |   movel([0.088081, -1.437744, -2.530560, -0.744085, 1.570796, 1.658878],accel_mss,speed_ms,0,blend_radius_m)
    |   movel([0.089883, -1.437273, -2.530932, -0.744184, 1.570796, 1.660679],accel_mss,speed_ms,0,blend_radius_m)
    |   movel([0.091685, -1.436804, -2.531302, -0.744283, 1.570796, 1.662481],accel_mss,speed_ms,0,blend_radius_m)
    |   movel([0.093488, -1.436337, -2.531669, -0.744382, 1.570796, 1.664284],accel_mss,speed_ms,0,blend_radius_m)
    |   movel([0.095833, -1.435725, -2.532151, -0.744512, 1.570796, 1.666629],accel_mss,speed_ms,0,blend_radius_m)
    |   speed_ms = 0.005
    |   # Splitting Linear movement in 6 (instruction 160: MoveL 140)
    |   movel([0.095833, -1.434329, -2.531529, -0.746531, 1.570796, 1.666629],accel_mss,speed_ms,0,blend_radius_m)
    |   movel([0.095833, -1.432937, -2.530904, -0.748548, 1.570796, 1.666629],accel_mss,speed_ms,0,blend_radius_m)
    |   movel([0.095833, -1.431548, -2.530279, -0.750562, 1.570796, 1.666629],accel_mss,speed_ms,0,blend_radius_m)
    |   movel([0.095833, -1.430163, -2.529651, -0.752575, 1.570796, 1.666629],accel_mss,speed_ms,0,blend_radius_m)
    |   movel([0.095833, -1.428783, -2.529022, -0.754585, 1.570796, 1.666629],accel_mss,speed_ms,0,blend_radius_m)
    |   movel([0.095833, -1.427406, -2.528391, -0.756593, 1.570796, 1.666629],accel_mss,speed_ms,0,blend_radius_m)
    |   speed_ms = 0.040
    |   # Splitting Linear movement in 16 (instruction 162: MoveL 141)
    |   movel([0.097717, -1.425761, -2.529667, -0.756962, 1.570796, 1.668513],accel_mss,speed_ms,0,blend_radius_m)
    |   movel([0.099607, -1.424113, -2.530940, -0.757335, 1.570796, 1.670403],accel_mss,speed_ms,0,blend_radius_m)
    |   movel([0.101503, -1.422463, -2.532212, -0.757714, 1.570796, 1.672299],accel_mss,speed_ms,0,blend_radius_m)
    |   movel([0.103405, -1.420810, -2.533482, -0.758097, 1.570796, 1.674201],accel_mss,speed_ms,0,blend_radius_m)
    |   movel([0.105313, -1.419154, -2.534750, -0.758485, 1.570796, 1.676110],accel_mss,speed_ms,0,blend_radius_m)
    |   movel([0.107228, -1.417495, -2.536016, -0.758878, 1.570796, 1.678024],accel_mss,speed_ms,0,blend_radius_m)
    |   movel([0.109148, -1.415834, -2.537280, -0.759275, 1.570796, 1.679945],accel_mss,speed_ms,0,blend_radius_m)
    |   movel([0.111075, -1.414170, -2.538542, -0.759677, 1.570796, 1.681872],accel_mss,speed_ms,0,blend_radius_m)
    |   movel([0.113008, -1.412502, -2.539802, -0.760084, 1.570796, 1.683805],accel_mss,speed_ms,0,blend_radius_m)
    |   movel([0.114947, -1.410833, -2.541061, -0.760496, 1.570796, 1.685744],accel_mss,speed_ms,0,blend_radius_m)
    |   movel([0.116893, -1.409160, -2.542317, -0.760912, 1.570796, 1.687689],accel_mss,speed_ms,0,blend_radius_m)
    |   movel([0.118845, -1.407484, -2.543571, -0.761334, 1.570796, 1.689641],accel_mss,speed_ms,0,blend_radius_m)
    |   movel([0.120803, -1.405806, -2.544823, -0.761760, 1.570796, 1.691599],accel_mss,speed_ms,0,blend_radius_m)
    |   movel([0.122767, -1.404124, -2.546074, -0.762191, 1.570796, 1.693563],accel_mss,speed_ms,0,blend_radius_m)
    |   movel([0.124738, -1.402440, -2.547322, -0.762627, 1.570796, 1.695534],accel_mss,speed_ms,0,blend_radius_m)
    |   movel([0.126715, -1.400753, -2.548568, -0.763068, 1.570796, 1.697511],accel_mss,speed_ms,0,blend_radius_m)
    |   speed_ms = 0.005
    |   # Splitting Linear movement in 4 (instruction 164: MoveL 142)
    |   movel([0.126715, -1.402869, -2.549542, -0.759978, 1.570796, 1.697511],accel_mss,speed_ms,0,blend_radius_m)
    |   movel([0.126715, -1.404994, -2.550512, -0.756883, 1.570796, 1.697511],accel_mss,speed_ms,0,blend_radius_m)
    |   movel([0.126715, -1.407128, -2.551479, -0.753783, 1.570796, 1.697511],accel_mss,speed_ms,0,blend_radius_m)
    |   movel([0.126715, -1.409271, -2.552441, -0.750677, 1.570796, 1.697511],accel_mss,speed_ms,0,blend_radius_m)
    |   speed_ms = 0.035
    |   # Splitting Linear movement in 4 (instruction 166: MoveL 143)
    |   movel([0.127916, -1.409507, -2.552265, -0.750617, 1.570796, 1.698712],accel_mss,speed_ms,0,blend_radius_m)
    |   movel([0.129116, -1.409743, -2.552088, -0.750557, 1.570796, 1.699912],accel_mss,speed_ms,0,blend_radius_m)
    |   movel([0.130314, -1.409982, -2.551910, -0.750497, 1.570796, 1.701111],accel_mss,speed_ms,0,blend_radius_m)
    |   movel([0.131512, -1.410222, -2.551730, -0.750437, 1.570796, 1.702308],accel_mss,speed_ms,0,blend_radius_m)
    |   # Splitting Linear movement in 10 (instruction 167: MoveL 144)
    |   movel([0.133306, -1.410596, -2.551450, -0.750343, 1.570796, 1.704102],accel_mss,speed_ms,0,blend_radius_m)
    |   movel([0.135097, -1.410974, -2.551167, -0.750248, 1.570796, 1.705893],accel_mss,speed_ms,0,blend_radius_m)
    |   movel([0.136885, -1.411355, -2.550881, -0.750153, 1.570796, 1.707681],accel_mss,speed_ms,0,blend_radius_m)
    |   movel([0.138670, -1.411739, -2.550592, -0.750057, 1.570796, 1.709467],accel_mss,speed_ms,0,blend_radius_m)
    |   movel([0.140452, -1.412127, -2.550301, -0.749961, 1.570796, 1.711249],accel_mss,speed_ms,0,blend_radius_m)
    |   movel([0.142231, -1.412519, -2.550007, -0.749863, 1.570796, 1.713028],accel_mss,speed_ms,0,blend_radius_m)
    |   movel([0.144008, -1.412914, -2.549709, -0.749766, 1.570796, 1.714804],accel_mss,speed_ms,0,blend_radius_m)
    |   movel([0.145781, -1.413312, -2.549409, -0.749667, 1.570796, 1.716577],accel_mss,speed_ms,0,blend_radius_m)
    |   movel([0.147551, -1.413714, -2.549107, -0.749568, 1.570796, 1.718347],accel_mss,speed_ms,0,blend_radius_m)
    |   movel([0.149318, -1.414120, -2.548801, -0.749468, 1.570796, 1.720114],accel_mss,speed_ms,0,blend_radius_m)
    |   movel([0.150561, -1.414495, -2.548517, -0.749376, 1.570796, 1.721357],accel_mss,speed_ms,0,blend_radius_m)
    |   movel([0.151594, -1.415065, -2.548087, -0.749237, 1.570796, 1.722391],accel_mss,speed_ms,0,blend_radius_m)
    |   movel([0.152000, -1.415449, -2.547797, -0.749143, 1.570796, 1.722797],accel_mss,speed_ms,0,blend_radius_m)
    |   movel([0.152314, -1.415910, -2.547448, -0.749031, 1.570796, 1.723110],accel_mss,speed_ms,0,blend_radius_m)
    |   movel([0.152520, -1.416461, -2.547030, -0.748897, 1.570796, 1.723316],accel_mss,speed_ms,0,blend_radius_m)
    |   movel([0.152610, -1.417112, -2.546537, -0.748740, 1.570796, 1.723406],accel_mss,speed_ms,0,blend_radius_m)
    |   movel([0.152506, -1.418145, -2.545752, -0.748492, 1.570796, 1.723302],accel_mss,speed_ms,0,blend_radius_m)
    |   movel([0.152142, -1.419177, -2.544967, -0.748246, 1.570796, 1.722939],accel_mss,speed_ms,0,blend_radius_m)
    |   movel([0.151550, -1.420173, -2.544207, -0.748009, 1.570796, 1.722346],accel_mss,speed_ms,0,blend_radius_m)
    |   movel([0.150755, -1.421109, -2.543492, -0.747788, 1.570796, 1.721551],accel_mss,speed_ms,0,blend_radius_m)
    |   movel([0.149785, -1.421957, -2.542843, -0.747590, 1.570796, 1.720581],accel_mss,speed_ms,0,blend_radius_m)
    |   movel([0.148671, -1.422685, -2.542285, -0.747420, 1.570796, 1.719467],accel_mss,speed_ms,0,blend_radius_m)
    |   movel([0.147440, -1.423265, -2.541839, -0.747285, 1.570796, 1.718236],accel_mss,speed_ms,0,blend_radius_m)
    |   movel([0.146116, -1.423673, -2.541526, -0.747190, 1.570796, 1.716912],accel_mss,speed_ms,0,blend_radius_m)
    |   # Splitting Linear movement in 8 (instruction 182: MoveL 159)
    |   movel([0.143924, -1.424158, -2.541153, -0.747078, 1.570796, 1.714720],accel_mss,speed_ms,0,blend_radius_m)
    |   movel([0.141732, -1.424646, -2.540777, -0.746966, 1.570796, 1.712528],accel_mss,speed_ms,0,blend_radius_m)
    |   movel([0.139541, -1.425138, -2.540398, -0.746853, 1.570796, 1.710337],accel_mss,speed_ms,0,blend_radius_m)
    |   movel([0.137350, -1.425633, -2.540016, -0.746740, 1.570796, 1.708146],accel_mss,speed_ms,0,blend_radius_m)
    |   movel([0.135160, -1.426132, -2.539631, -0.746626, 1.570796, 1.705956],accel_mss,speed_ms,0,blend_radius_m)
    |   movel([0.132971, -1.426633, -2.539243, -0.746512, 1.570796, 1.703767],accel_mss,speed_ms,0,blend_radius_m)
    |   movel([0.130782, -1.427139, -2.538852, -0.746398, 1.570796, 1.701579],accel_mss,speed_ms,0,blend_radius_m)
    |   movel([0.128595, -1.427647, -2.538459, -0.746283, 1.570796, 1.699391],accel_mss,speed_ms,0,blend_radius_m)
    |   movel([0.127707, -1.427936, -2.538235, -0.746218, 1.570796, 1.698503],accel_mss,speed_ms,0,blend_radius_m)
    |   movel([0.127123, -1.428343, -2.537919, -0.746127, 1.570796, 1.697919],accel_mss,speed_ms,0,blend_radius_m)
    |   movel([0.126772, -1.428905, -2.537483, -0.746001, 1.570796, 1.697568],accel_mss,speed_ms,0,blend_radius_m)
    |   movel([0.126581, -1.429656, -2.536900, -0.745834, 1.570796, 1.697378],accel_mss,speed_ms,0,blend_radius_m)
    |   movel([0.126552, -1.430104, -2.536551, -0.745734, 1.570796, 1.697348],accel_mss,speed_ms,0,blend_radius_m)
    |   movel([0.126785, -1.430619, -2.536150, -0.745620, 1.570796, 1.697581],accel_mss,speed_ms,0,blend_radius_m)
    |   movel([0.127017, -1.430723, -2.536068, -0.745597, 1.570796, 1.697813],accel_mss,speed_ms,0,blend_radius_m)
    |   movel([0.127657, -1.430719, -2.536072, -0.745598, 1.570796, 1.698454],accel_mss,speed_ms,0,blend_radius_m)
    |   movel([0.128440, -1.430554, -2.536200, -0.745635, 1.570796, 1.699236],accel_mss,speed_ms,0,blend_radius_m)
    |   # Splitting Linear movement in 8 (instruction 192: MoveL 169)
    |   movel([0.130720, -1.430012, -2.536622, -0.745754, 1.570796, 1.701517],accel_mss,speed_ms,0,blend_radius_m)
    |   movel([0.133001, -1.429474, -2.537041, -0.745874, 1.570796, 1.703798],accel_mss,speed_ms,0,blend_radius_m)
    |   movel([0.135283, -1.428939, -2.537457, -0.745993, 1.570796, 1.706080],accel_mss,speed_ms,0,blend_radius_m)
    |   movel([0.137566, -1.428408, -2.537869, -0.746112, 1.570796, 1.708362],accel_mss,speed_ms,0,blend_radius_m)
    |   movel([0.139850, -1.427880, -2.538278, -0.746231, 1.570796, 1.710646],accel_mss,speed_ms,0,blend_radius_m)
    |   movel([0.142134, -1.427357, -2.538684, -0.746349, 1.570796, 1.712930],accel_mss,speed_ms,0,blend_radius_m)
    |   movel([0.144419, -1.426836, -2.539086, -0.746466, 1.570796, 1.715215],accel_mss,speed_ms,0,blend_radius_m)
    |   movel([0.146705, -1.426320, -2.539486, -0.746583, 1.570796, 1.717501],accel_mss,speed_ms,0,blend_radius_m)
    |   movel([0.147624, -1.426053, -2.539692, -0.746644, 1.570796, 1.718420],accel_mss,speed_ms,0,blend_radius_m)
    |   movel([0.149504, -1.425233, -2.540325, -0.746831, 1.570796, 1.720300],accel_mss,speed_ms,0,blend_radius_m)
    |   movel([0.150393, -1.424714, -2.540724, -0.746950, 1.570796, 1.721189],accel_mss,speed_ms,0,blend_radius_m)
    |   movel([0.151559, -1.423902, -2.541350, -0.747138, 1.570796, 1.722356],accel_mss,speed_ms,0,blend_radius_m)
    |   movel([0.152591, -1.423034, -2.542016, -0.747338, 1.570796, 1.723388],accel_mss,speed_ms,0,blend_radius_m)
    |   movel([0.153490, -1.422118, -2.542719, -0.747552, 1.570796, 1.724287],accel_mss,speed_ms,0,blend_radius_m)
    |   movel([0.154255, -1.421155, -2.543456, -0.747777, 1.570796, 1.725052],accel_mss,speed_ms,0,blend_radius_m)
    |   movel([0.154893, -1.420150, -2.544225, -0.748015, 1.570796, 1.725689],accel_mss,speed_ms,0,blend_radius_m)
    |   movel([0.155401, -1.419104, -2.545022, -0.748263, 1.570796, 1.726197],accel_mss,speed_ms,0,blend_radius_m)
    |   movel([0.155784, -1.418024, -2.545844, -0.748521, 1.570796, 1.726580],accel_mss,speed_ms,0,blend_radius_m)
    |   movel([0.156043, -1.416910, -2.546690, -0.748789, 1.570796, 1.726840],accel_mss,speed_ms,0,blend_radius_m)
    |   movel([0.156154, -1.415805, -2.547528, -0.749057, 1.570796, 1.726951],accel_mss,speed_ms,0,blend_radius_m)
    |   movel([0.156082, -1.414817, -2.548275, -0.749298, 1.570796, 1.726878],accel_mss,speed_ms,0,blend_radius_m)
    |   movel([0.155834, -1.413946, -2.548932, -0.749511, 1.570796, 1.726630],accel_mss,speed_ms,0,blend_radius_m)
    |   movel([0.155422, -1.413191, -2.549501, -0.749697, 1.570796, 1.726218],accel_mss,speed_ms,0,blend_radius_m)
    |   movel([0.154853, -1.412548, -2.549985, -0.749856, 1.570796, 1.725650],accel_mss,speed_ms,0,blend_radius_m)
    |   movel([0.154139, -1.412020, -2.550382, -0.749987, 1.570796, 1.724936],accel_mss,speed_ms,0,blend_radius_m)
    |   movel([0.153287, -1.411601, -2.550696, -0.750092, 1.570796, 1.724083],accel_mss,speed_ms,0,blend_radius_m)
    |   movel([0.152307, -1.411291, -2.550929, -0.750169, 1.570796, 1.723103],accel_mss,speed_ms,0,blend_radius_m)
    |   # Splitting Linear movement in 14 (instruction 212: MoveL 189)
    |   movel([0.150360, -1.410836, -2.551271, -0.750283, 1.570796, 1.721157],accel_mss,speed_ms,0,blend_radius_m)
    |   movel([0.148410, -1.410385, -2.551608, -0.750396, 1.570796, 1.719206],accel_mss,speed_ms,0,blend_radius_m)
    |   movel([0.146456, -1.409938, -2.551943, -0.750508, 1.570796, 1.717252],accel_mss,speed_ms,0,blend_radius_m)
    |   movel([0.144498, -1.409495, -2.552274, -0.750620, 1.570796, 1.715294],accel_mss,speed_ms,0,blend_radius_m)
    |   movel([0.142537, -1.409057, -2.552601, -0.750731, 1.570796, 1.713333],accel_mss,speed_ms,0,blend_radius_m)
    |   movel([0.140571, -1.408623, -2.552926, -0.750841, 1.570796, 1.711368],accel_mss,speed_ms,0,blend_radius_m)
    |   movel([0.138603, -1.408193, -2.553246, -0.750950, 1.570796, 1.709399],accel_mss,speed_ms,0,blend_radius_m)
    |   movel([0.136630, -1.407767, -2.553564, -0.751059, 1.570796, 1.707426],accel_mss,speed_ms,0,blend_radius_m)
    |   movel([0.134654, -1.407345, -2.553877, -0.751166, 1.570796, 1.705450],accel_mss,speed_ms,0,blend_radius_m)
    |   movel([0.132674, -1.406928, -2.554188, -0.751273, 1.570796, 1.703470],accel_mss,speed_ms,0,blend_radius_m)
    |   movel([0.130690, -1.406515, -2.554495, -0.751379, 1.570796, 1.701486],accel_mss,speed_ms,0,blend_radius_m)
    |   movel([0.128703, -1.406107, -2.554798, -0.751484, 1.570796, 1.699499],accel_mss,speed_ms,0,blend_radius_m)
    |   movel([0.126712, -1.405702, -2.555099, -0.751588, 1.570796, 1.697508],accel_mss,speed_ms,0,blend_radius_m)
    |   movel([0.124717, -1.405302, -2.555395, -0.751692, 1.570796, 1.695514],accel_mss,speed_ms,0,blend_radius_m)
    |   movel([0.123823, -1.405439, -2.555294, -0.751656, 1.570796, 1.694619],accel_mss,speed_ms,0,blend_radius_m)
    |   # Splitting Linear movement in 16 (instruction 214: MoveL 191)
    |   movel([0.123525, -1.407503, -2.553760, -0.751126, 1.570796, 1.694321],accel_mss,speed_ms,0,blend_radius_m)
    |   movel([0.123228, -1.409561, -2.552225, -0.750603, 1.570796, 1.694025],accel_mss,speed_ms,0,blend_radius_m)
    |   movel([0.122933, -1.411613, -2.550687, -0.750089, 1.570796, 1.693729],accel_mss,speed_ms,0,blend_radius_m)
    |   movel([0.122639, -1.413658, -2.549149, -0.749582, 1.570796, 1.693436],accel_mss,speed_ms,0,blend_radius_m)
    |   movel([0.122347, -1.415698, -2.547609, -0.749083, 1.570796, 1.693143],accel_mss,speed_ms,0,blend_radius_m)
    |   movel([0.122056, -1.417731, -2.546067, -0.748591, 1.570796, 1.692852],accel_mss,speed_ms,0,blend_radius_m)
    |   movel([0.121766, -1.419758, -2.544524, -0.748107, 1.570796, 1.692563],accel_mss,speed_ms,0,blend_radius_m)
    |   movel([0.121478, -1.421779, -2.542979, -0.747631, 1.570796, 1.692275],accel_mss,speed_ms,0,blend_radius_m)
    |   movel([0.121191, -1.423794, -2.541433, -0.747162, 1.570796, 1.691988],accel_mss,speed_ms,0,blend_radius_m)
    |   movel([0.120906, -1.425803, -2.539885, -0.746701, 1.570796, 1.691702],accel_mss,speed_ms,0,blend_radius_m)
    |   movel([0.120622, -1.427806, -2.538335, -0.746247, 1.570796, 1.691418],accel_mss,speed_ms,0,blend_radius_m)
    |   movel([0.120339, -1.429804, -2.536785, -0.745801, 1.570796, 1.691136],accel_mss,speed_ms,0,blend_radius_m)
    |   movel([0.120058, -1.431795, -2.535232, -0.745362, 1.570796, 1.690854],accel_mss,speed_ms,0,blend_radius_m)
    |   movel([0.119778, -1.433781, -2.533679, -0.744930, 1.570796, 1.690574],accel_mss,speed_ms,0,blend_radius_m)
    |   movel([0.119499, -1.435761, -2.532124, -0.744505, 1.570796, 1.690295],accel_mss,speed_ms,0,blend_radius_m)
    |   movel([0.119222, -1.437735, -2.530567, -0.744087, 1.570796, 1.690018],accel_mss,speed_ms,0,blend_radius_m)
    |   movel([0.119226, -1.438624, -2.529864, -0.743901, 1.570796, 1.690023],accel_mss,speed_ms,0,blend_radius_m)
    |   movel([0.119359, -1.438887, -2.529655, -0.743846, 1.570796, 1.690155],accel_mss,speed_ms,0,blend_radius_m)
    |   movel([0.119573, -1.439046, -2.529530, -0.743813, 1.570796, 1.690369],accel_mss,speed_ms,0,blend_radius_m)
    |   movel([0.120234, -1.439103, -2.529485, -0.743801, 1.570796, 1.691030],accel_mss,speed_ms,0,blend_radius_m)
    |   movel([0.121194, -1.438890, -2.529653, -0.743846, 1.570796, 1.691990],accel_mss,speed_ms,0,blend_radius_m)
    |   movel([0.121707, -1.438702, -2.529802, -0.743885, 1.570796, 1.692504],accel_mss,speed_ms,0,blend_radius_m)
    |   movel([0.122081, -1.438478, -2.529979, -0.743931, 1.570796, 1.692878],accel_mss,speed_ms,0,blend_radius_m)
    |   movel([0.122340, -1.438225, -2.530179, -0.743984, 1.570796, 1.693137],accel_mss,speed_ms,0,blend_radius_m)
    |   movel([0.122506, -1.437952, -2.530395, -0.744042, 1.570796, 1.693302],accel_mss,speed_ms,0,blend_radius_m)
    |   movel([0.122653, -1.437362, -2.530861, -0.744166, 1.570796, 1.693450],accel_mss,speed_ms,0,blend_radius_m)
    |   movel([0.122716, -1.436766, -2.531332, -0.744291, 1.570796, 1.693512],accel_mss,speed_ms,0,blend_radius_m)
    |   # Splitting Linear movement in 14 (instruction 226: MoveL 203)
    |   movel([0.122993, -1.434839, -2.532849, -0.744702, 1.570796, 1.693789],accel_mss,speed_ms,0,blend_radius_m)
    |   movel([0.123271, -1.432906, -2.534364, -0.745119, 1.570796, 1.694068],accel_mss,speed_ms,0,blend_radius_m)
    |   movel([0.123551, -1.430967, -2.535878, -0.745543, 1.570796, 1.694347],accel_mss,speed_ms,0,blend_radius_m)
    |   movel([0.123832, -1.429023, -2.537391, -0.745974, 1.570796, 1.694628],accel_mss,speed_ms,0,blend_radius_m)
    |   movel([0.124114, -1.427074, -2.538903, -0.746412, 1.570796, 1.694911],accel_mss,speed_ms,0,blend_radius_m)
    |   movel([0.124398, -1.425119, -2.540413, -0.746858, 1.570796, 1.695194],accel_mss,speed_ms,0,blend_radius_m)
    |   movel([0.124683, -1.423158, -2.541921, -0.747310, 1.570796, 1.695479],accel_mss,speed_ms,0,blend_radius_m)
    |   movel([0.124969, -1.421192, -2.543428, -0.747769, 1.570796, 1.695765],accel_mss,speed_ms,0,blend_radius_m)
    |   movel([0.125257, -1.419219, -2.544934, -0.748235, 1.570796, 1.696053],accel_mss,speed_ms,0,blend_radius_m)
    |   movel([0.125546, -1.417242, -2.546439, -0.748709, 1.570796, 1.696342],accel_mss,speed_ms,0,blend_radius_m)
    |   movel([0.125836, -1.415258, -2.547941, -0.749190, 1.570796, 1.696632],accel_mss,speed_ms,0,blend_radius_m)
    |   movel([0.126128, -1.413268, -2.549443, -0.749678, 1.570796, 1.696924],accel_mss,speed_ms,0,blend_radius_m)
    |   movel([0.126421, -1.411273, -2.550943, -0.750174, 1.570796, 1.697217],accel_mss,speed_ms,0,blend_radius_m)
    |   movel([0.126715, -1.409271, -2.552441, -0.750677, 1.570796, 1.697511],accel_mss,speed_ms,0,blend_radius_m)
    |   movel([0.128744, -1.409671, -2.552143, -0.750576, 1.570796, 1.699541],accel_mss,speed_ms,0,blend_radius_m)
    |   speed_ms = 0.005
    |   # Splitting Linear movement in 6 (instruction 229: MoveL 205)
    |   movel([0.128744, -1.408241, -2.551502, -0.752646, 1.570796, 1.699541],accel_mss,speed_ms,0,blend_radius_m)
    |   movel([0.128744, -1.406816, -2.550859, -0.754714, 1.570796, 1.699541],accel_mss,speed_ms,0,blend_radius_m)
    |   movel([0.128744, -1.405394, -2.550214, -0.756780, 1.570796, 1.699541],accel_mss,speed_ms,0,blend_radius_m)
    |   movel([0.128744, -1.403977, -2.549568, -0.758843, 1.570796, 1.699541],accel_mss,speed_ms,0,blend_radius_m)
    |   movel([0.128744, -1.402564, -2.548921, -0.760904, 1.570796, 1.699541],accel_mss,speed_ms,0,blend_radius_m)
    |   movel([0.128744, -1.401155, -2.548271, -0.762962, 1.570796, 1.699541],accel_mss,speed_ms,0,blend_radius_m)
    |   speed_ms = 0.040
    |   # Splitting Linear movement in 12 (instruction 231: MoveL 206)
    |   movel([0.127186, -1.400512, -2.548746, -0.763131, 1.570796, 1.697982],accel_mss,speed_ms,0,blend_radius_m)
    |   movel([0.125624, -1.399871, -2.549218, -0.763300, 1.570796, 1.696420],accel_mss,speed_ms,0,blend_radius_m)
    |   movel([0.124058, -1.399233, -2.549688, -0.763469, 1.570796, 1.694855],accel_mss,speed_ms,0,blend_radius_m)
    |   movel([0.122489, -1.398597, -2.550155, -0.763637, 1.570796, 1.693286],accel_mss,speed_ms,0,blend_radius_m)
    |   movel([0.120917, -1.397964, -2.550619, -0.763806, 1.570796, 1.691713],accel_mss,speed_ms,0,blend_radius_m)
    |   movel([0.119341, -1.397334, -2.551081, -0.763974, 1.570796, 1.690137],accel_mss,speed_ms,0,blend_radius_m)
    |   movel([0.117762, -1.396707, -2.551540, -0.764142, 1.570796, 1.688558],accel_mss,speed_ms,0,blend_radius_m)
    |   movel([0.116179, -1.396082, -2.551997, -0.764310, 1.570796, 1.686975],accel_mss,speed_ms,0,blend_radius_m)
    |   movel([0.114593, -1.395461, -2.552451, -0.764478, 1.570796, 1.685389],accel_mss,speed_ms,0,blend_radius_m)
    |   movel([0.113003, -1.394842, -2.552902, -0.764645, 1.570796, 1.683799],accel_mss,speed_ms,0,blend_radius_m)
    |   movel([0.111410, -1.394225, -2.553351, -0.764812, 1.570796, 1.682206],accel_mss,speed_ms,0,blend_radius_m)
    |   movel([0.109813, -1.393612, -2.553797, -0.764980, 1.570796, 1.680610],accel_mss,speed_ms,0,blend_radius_m)
    |   speed_ms = 0.005
    |   # Splitting Linear movement in 4 (instruction 233: MoveL 207)
    |   movel([0.109813, -1.395740, -2.554779, -0.761870, 1.570796, 1.680610],accel_mss,speed_ms,0,blend_radius_m)
    |   movel([0.109813, -1.397878, -2.555757, -0.758754, 1.570796, 1.680610],accel_mss,speed_ms,0,blend_radius_m)
    |   movel([0.109813, -1.400026, -2.556731, -0.755633, 1.570796, 1.680610],accel_mss,speed_ms,0,blend_radius_m)
    |   movel([0.109813, -1.402182, -2.557701, -0.752506, 1.570796, 1.680610],accel_mss,speed_ms,0,blend_radius_m)
    |   speed_ms = 0.035
    |   movel([0.111645, -1.402395, -2.557544, -0.752450, 1.570796, 1.682442],accel_mss,speed_ms,0,blend_radius_m)
    |   movel([0.112194, -1.402556, -2.557426, -0.752408, 1.570796, 1.682991],accel_mss,speed_ms,0,blend_radius_m)
    |   movel([0.112546, -1.402800, -2.557245, -0.752343, 1.570796, 1.683343],accel_mss,speed_ms,0,blend_radius_m)
    |   movel([0.112731, -1.403170, -2.556973, -0.752247, 1.570796, 1.683527],accel_mss,speed_ms,0,blend_radius_m)
    |   movel([0.112779, -1.403700, -2.556581, -0.752108, 1.570796, 1.683575],accel_mss,speed_ms,0,blend_radius_m)
    |   movel([0.112607, -1.405387, -2.555333, -0.751670, 1.570796, 1.683404],accel_mss,speed_ms,0,blend_radius_m)
    |   # Splitting Linear movement in 18 (instruction 241: MoveL 214)
    |   movel([0.112349, -1.407375, -2.553855, -0.751158, 1.570796, 1.683145],accel_mss,speed_ms,0,blend_radius_m)
    |   movel([0.112092, -1.409358, -2.552376, -0.750655, 1.570796, 1.682888],accel_mss,speed_ms,0,blend_radius_m)
    |   movel([0.111836, -1.411336, -2.550896, -0.750158, 1.570796, 1.682632],accel_mss,speed_ms,0,blend_radius_m)
    |   movel([0.111581, -1.413307, -2.549414, -0.749668, 1.570796, 1.682377],accel_mss,speed_ms,0,blend_radius_m)
    |   movel([0.111328, -1.415273, -2.547930, -0.749186, 1.570796, 1.682124],accel_mss,speed_ms,0,blend_radius_m)
    |   movel([0.111075, -1.417233, -2.546445, -0.748711, 1.570796, 1.681871],accel_mss,speed_ms,0,blend_radius_m)
    |   movel([0.110824, -1.419187, -2.544959, -0.748243, 1.570796, 1.681620],accel_mss,speed_ms,0,blend_radius_m)
    |   movel([0.110574, -1.421136, -2.543471, -0.747782, 1.570796, 1.681370],accel_mss,speed_ms,0,blend_radius_m)
    |   movel([0.110325, -1.423079, -2.541982, -0.747328, 1.570796, 1.681121],accel_mss,speed_ms,0,blend_radius_m)
    |   movel([0.110077, -1.425017, -2.540491, -0.746881, 1.570796, 1.680873],accel_mss,speed_ms,0,blend_radius_m)
    |   movel([0.109831, -1.426949, -2.538999, -0.746441, 1.570796, 1.680627],accel_mss,speed_ms,0,blend_radius_m)
    |   movel([0.109585, -1.428875, -2.537506, -0.746007, 1.570796, 1.680381],accel_mss,speed_ms,0,blend_radius_m)
    |   movel([0.109341, -1.430797, -2.536011, -0.745581, 1.570796, 1.680137],accel_mss,speed_ms,0,blend_radius_m)
    |   movel([0.109097, -1.432713, -2.534515, -0.745161, 1.570796, 1.679894],accel_mss,speed_ms,0,blend_radius_m)
    |   movel([0.108855, -1.434624, -2.533017, -0.744748, 1.570796, 1.679652],accel_mss,speed_ms,0,blend_radius_m)
    |   movel([0.108614, -1.436529, -2.531518, -0.744342, 1.570796, 1.679411],accel_mss,speed_ms,0,blend_radius_m)
    |   movel([0.108374, -1.438429, -2.530018, -0.743942, 1.570796, 1.679171],accel_mss,speed_ms,0,blend_radius_m)
    |   movel([0.108135, -1.440324, -2.528516, -0.743548, 1.570796, 1.678932],accel_mss,speed_ms,0,blend_radius_m)
    |   movel([0.107909, -1.441254, -2.527777, -0.743357, 1.570796, 1.678706],accel_mss,speed_ms,0,blend_radius_m)
    |   movel([0.107474, -1.441934, -2.527237, -0.743219, 1.570796, 1.678271],accel_mss,speed_ms,0,blend_radius_m)
    |   movel([0.107164, -1.442179, -2.527041, -0.743169, 1.570796, 1.677960],accel_mss,speed_ms,0,blend_radius_m)
    |   movel([0.106790, -1.442362, -2.526896, -0.743132, 1.570796, 1.677586],accel_mss,speed_ms,0,blend_radius_m)
    |   movel([0.105823, -1.442532, -2.526760, -0.743097, 1.570796, 1.676619],accel_mss,speed_ms,0,blend_radius_m)
    |   movel([0.105416, -1.442467, -2.526812, -0.743110, 1.570796, 1.676213],accel_mss,speed_ms,0,blend_radius_m)
    |   movel([0.105033, -1.442273, -2.526966, -0.743150, 1.570796, 1.675829],accel_mss,speed_ms,0,blend_radius_m)
    |   movel([0.104755, -1.442000, -2.527183, -0.743205, 1.570796, 1.675551],accel_mss,speed_ms,0,blend_radius_m)
    |   movel([0.104666, -1.441699, -2.527424, -0.743267, 1.570796, 1.675462],accel_mss,speed_ms,0,blend_radius_m)
    |   # Splitting Linear movement in 20 (instruction 251: MoveL 224)
    |   movel([0.104899, -1.439799, -2.528933, -0.743657, 1.570796, 1.675695],accel_mss,speed_ms,0,blend_radius_m)
    |   movel([0.105133, -1.437894, -2.530441, -0.744054, 1.570796, 1.675929],accel_mss,speed_ms,0,blend_radius_m)
    |   movel([0.105367, -1.435984, -2.531948, -0.744457, 1.570796, 1.676164],accel_mss,speed_ms,0,blend_radius_m)
    |   movel([0.105603, -1.434069, -2.533453, -0.744867, 1.570796, 1.676400],accel_mss,speed_ms,0,blend_radius_m)
    |   movel([0.105840, -1.432148, -2.534957, -0.745284, 1.570796, 1.676637],accel_mss,speed_ms,0,blend_radius_m)
    |   movel([0.106079, -1.430222, -2.536459, -0.745708, 1.570796, 1.676875],accel_mss,speed_ms,0,blend_radius_m)
    |   movel([0.106318, -1.428291, -2.537960, -0.746138, 1.570796, 1.677114],accel_mss,speed_ms,0,blend_radius_m)
    |   movel([0.106558, -1.426354, -2.539459, -0.746576, 1.570796, 1.677355],accel_mss,speed_ms,0,blend_radius_m)
    |   movel([0.106800, -1.424411, -2.540958, -0.747020, 1.570796, 1.677596],accel_mss,speed_ms,0,blend_radius_m)
    |   movel([0.107042, -1.422464, -2.542454, -0.747471, 1.570796, 1.677839],accel_mss,speed_ms,0,blend_radius_m)
    |   movel([0.107286, -1.420510, -2.543949, -0.747929, 1.570796, 1.678082],accel_mss,speed_ms,0,blend_radius_m)
    |   movel([0.107531, -1.418551, -2.545443, -0.748395, 1.570796, 1.678327],accel_mss,speed_ms,0,blend_radius_m)
    |   movel([0.107777, -1.416586, -2.546936, -0.748867, 1.570796, 1.678573],accel_mss,speed_ms,0,blend_radius_m)
    |   movel([0.108024, -1.414616, -2.548426, -0.749347, 1.570796, 1.678820],accel_mss,speed_ms,0,blend_radius_m)
    |   movel([0.108272, -1.412640, -2.549916, -0.749833, 1.570796, 1.679069],accel_mss,speed_ms,0,blend_radius_m)
    |   movel([0.108522, -1.410658, -2.551404, -0.750327, 1.570796, 1.679318],accel_mss,speed_ms,0,blend_radius_m)
    |   movel([0.108773, -1.408670, -2.552890, -0.750829, 1.570796, 1.679569],accel_mss,speed_ms,0,blend_radius_m)
    |   movel([0.109024, -1.406676, -2.554375, -0.751338, 1.570796, 1.679821],accel_mss,speed_ms,0,blend_radius_m)
    |   movel([0.109278, -1.404677, -2.555859, -0.751854, 1.570796, 1.680074],accel_mss,speed_ms,0,blend_radius_m)
    |   movel([0.109532, -1.402671, -2.557341, -0.752377, 1.570796, 1.680328],accel_mss,speed_ms,0,blend_radius_m)
    |   movel([0.109813, -1.402182, -2.557701, -0.752506, 1.570796, 1.680610],accel_mss,speed_ms,0,blend_radius_m)
    |   movel([0.111645, -1.402395, -2.557544, -0.752450, 1.570796, 1.682442],accel_mss,speed_ms,0,blend_radius_m)
    |   movel([0.111918, -1.402475, -2.557485, -0.752429, 1.570796, 1.682714],accel_mss,speed_ms,0,blend_radius_m)
    |   speed_ms = 0.005
    |   # Splitting Linear movement in 6 (instruction 256: MoveL 228)
    |   movel([0.111918, -1.401036, -2.556839, -0.754514, 1.570796, 1.682714],accel_mss,speed_ms,0,blend_radius_m)
    |   movel([0.111918, -1.399602, -2.556191, -0.756596, 1.570796, 1.682714],accel_mss,speed_ms,0,blend_radius_m)
    |   movel([0.111918, -1.398172, -2.555542, -0.758676, 1.570796, 1.682714],accel_mss,speed_ms,0,blend_radius_m)
    |   movel([0.111918, -1.396746, -2.554890, -0.760753, 1.570796, 1.682714],accel_mss,speed_ms,0,blend_radius_m)
    |   movel([0.111918, -1.395324, -2.554238, -0.762827, 1.570796, 1.682714],accel_mss,speed_ms,0,blend_radius_m)
    |   movel([0.111918, -1.393907, -2.553583, -0.764899, 1.570796, 1.682714],accel_mss,speed_ms,0,blend_radius_m)
    |   speed_ms = 0.040
    |   # Splitting Linear movement in 8 (instruction 258: MoveL 229)
    |   movel([0.112997, -1.392012, -2.554959, -0.765418, 1.570796, 1.683793],accel_mss,speed_ms,0,blend_radius_m)
    |   movel([0.114080, -1.390112, -2.556333, -0.765944, 1.570796, 1.684876],accel_mss,speed_ms,0,blend_radius_m)
    |   movel([0.115168, -1.388206, -2.557707, -0.766476, 1.570796, 1.685964],accel_mss,speed_ms,0,blend_radius_m)
    |   movel([0.116260, -1.386295, -2.559079, -0.767015, 1.570796, 1.687057],accel_mss,speed_ms,0,blend_radius_m)
    |   movel([0.117357, -1.384378, -2.560450, -0.767561, 1.570796, 1.688154],accel_mss,speed_ms,0,blend_radius_m)
    |   movel([0.118459, -1.382455, -2.561820, -0.768114, 1.570796, 1.689255],accel_mss,speed_ms,0,blend_radius_m)
    |   movel([0.119565, -1.380526, -2.563189, -0.768674, 1.570796, 1.690361],accel_mss,speed_ms,0,blend_radius_m)
    |   movel([0.120675, -1.378592, -2.564556, -0.769241, 1.570796, 1.691472],accel_mss,speed_ms,0,blend_radius_m)
    |   speed_ms = 0.005
    |   # Splitting Linear movement in 4 (instruction 260: MoveL 230)
    |   movel([0.120675, -1.380746, -2.565554, -0.766089, 1.570796, 1.691472],accel_mss,speed_ms,0,blend_radius_m)
    |   movel([0.120675, -1.382911, -2.566548, -0.762930, 1.570796, 1.691472],accel_mss,speed_ms,0,blend_radius_m)
    |   movel([0.120675, -1.385085, -2.567538, -0.759765, 1.570796, 1.691472],accel_mss,speed_ms,0,blend_radius_m)
    |   movel([0.120675, -1.387270, -2.568525, -0.756595, 1.570796, 1.691472],accel_mss,speed_ms,0,blend_radius_m)
    |   speed_ms = 0.035
    |   # Splitting Linear movement in 22 (instruction 262: MoveL 231)
    |   movel([0.122721, -1.387699, -2.568217, -0.756472, 1.570796, 1.693518],accel_mss,speed_ms,0,blend_radius_m)
    |   movel([0.124763, -1.388134, -2.567906, -0.756349, 1.570796, 1.695560],accel_mss,speed_ms,0,blend_radius_m)
    |   movel([0.126802, -1.388572, -2.567592, -0.756225, 1.570796, 1.697598],accel_mss,speed_ms,0,blend_radius_m)
    |   movel([0.128836, -1.389016, -2.567274, -0.756099, 1.570796, 1.699632],accel_mss,speed_ms,0,blend_radius_m)
    |   movel([0.130866, -1.389464, -2.566953, -0.755973, 1.570796, 1.701662],accel_mss,speed_ms,0,blend_radius_m)
    |   movel([0.132892, -1.389916, -2.566627, -0.755845, 1.570796, 1.703688],accel_mss,speed_ms,0,blend_radius_m)
    |   movel([0.134914, -1.390373, -2.566299, -0.755717, 1.570796, 1.705710],accel_mss,speed_ms,0,blend_radius_m)
    |   movel([0.136932, -1.390835, -2.565967, -0.755588, 1.570796, 1.707728],accel_mss,speed_ms,0,blend_radius_m)
    |   movel([0.138946, -1.391301, -2.565631, -0.755457, 1.570796, 1.709742],accel_mss,speed_ms,0,blend_radius_m)
    |   movel([0.140956, -1.391771, -2.565291, -0.755326, 1.570796, 1.711753],accel_mss,speed_ms,0,blend_radius_m)
    |   movel([0.142962, -1.392246, -2.564949, -0.755194, 1.570796, 1.713759],accel_mss,speed_ms,0,blend_radius_m)
    |   movel([0.144964, -1.392726, -2.564602, -0.755061, 1.570796, 1.715760],accel_mss,speed_ms,0,blend_radius_m)
    |   movel([0.146962, -1.393210, -2.564252, -0.754927, 1.570796, 1.717758],accel_mss,speed_ms,0,blend_radius_m)
    |   movel([0.148956, -1.393698, -2.563899, -0.754792, 1.570796, 1.719752],accel_mss,speed_ms,0,blend_radius_m)
    |   movel([0.150946, -1.394191, -2.563542, -0.754657, 1.570796, 1.721742],accel_mss,speed_ms,0,blend_radius_m)
    |   movel([0.152931, -1.394688, -2.563181, -0.754520, 1.570796, 1.723728],accel_mss,speed_ms,0,blend_radius_m)
    |   movel([0.154913, -1.395189, -2.562817, -0.754383, 1.570796, 1.725709],accel_mss,speed_ms,0,blend_radius_m)
    |   movel([0.156890, -1.395695, -2.562449, -0.754245, 1.570796, 1.727687],accel_mss,speed_ms,0,blend_radius_m)
    |   movel([0.158864, -1.396205, -2.562078, -0.754106, 1.570796, 1.729660],accel_mss,speed_ms,0,blend_radius_m)
    |   movel([0.160833, -1.396719, -2.561704, -0.753966, 1.570796, 1.731629],accel_mss,speed_ms,0,blend_radius_m)
    |   movel([0.162798, -1.397238, -2.561326, -0.753825, 1.570796, 1.733594],accel_mss,speed_ms,0,blend_radius_m)
    |   movel([0.164759, -1.397761, -2.560944, -0.753684, 1.570796, 1.735555],accel_mss,speed_ms,0,blend_radius_m)
    |   movel([0.166439, -1.398301, -2.560549, -0.753539, 1.570796, 1.737236],accel_mss,speed_ms,0,blend_radius_m)
    |   movel([0.167973, -1.398997, -2.560040, -0.753352, 1.570796, 1.738769],accel_mss,speed_ms,0,blend_radius_m)
    |   movel([0.169359, -1.399836, -2.559425, -0.753127, 1.570796, 1.740155],accel_mss,speed_ms,0,blend_radius_m)
    |   movel([0.170595, -1.400812, -2.558709, -0.752868, 1.570796, 1.741391],accel_mss,speed_ms,0,blend_radius_m)
    |   movel([0.171678, -1.401913, -2.557899, -0.752577, 1.570796, 1.742474],accel_mss,speed_ms,0,blend_radius_m)
    |   movel([0.172602, -1.403132, -2.557000, -0.752256, 1.570796, 1.743398],accel_mss,speed_ms,0,blend_radius_m)
    |   movel([0.173367, -1.404460, -2.556019, -0.751910, 1.570796, 1.744164],accel_mss,speed_ms,0,blend_radius_m)
    |   movel([0.173972, -1.405884, -2.554964, -0.751541, 1.570796, 1.744768],accel_mss,speed_ms,0,blend_radius_m)
    |   movel([0.174412, -1.407397, -2.553839, -0.751153, 1.570796, 1.745208],accel_mss,speed_ms,0,blend_radius_m)
    |   movel([0.174688, -1.408991, -2.552651, -0.750747, 1.570796, 1.745484],accel_mss,speed_ms,0,blend_radius_m)
    |   movel([0.174793, -1.410653, -2.551407, -0.750329, 1.570796, 1.745589],accel_mss,speed_ms,0,blend_radius_m)
    |   movel([0.174728, -1.412378, -2.550112, -0.749898, 1.570796, 1.745525],accel_mss,speed_ms,0,blend_radius_m)
    |   movel([0.174493, -1.414156, -2.548773, -0.749459, 1.570796, 1.745289],accel_mss,speed_ms,0,blend_radius_m)
    |   movel([0.174082, -1.415977, -2.547397, -0.749015, 1.570796, 1.744878],accel_mss,speed_ms,0,blend_radius_m)
    |   movel([0.173496, -1.417834, -2.545989, -0.748566, 1.570796, 1.744293],accel_mss,speed_ms,0,blend_radius_m)
    |   movel([0.172732, -1.419716, -2.544556, -0.748117, 1.570796, 1.743529],accel_mss,speed_ms,0,blend_radius_m)
    |   movel([0.171793, -1.421622, -2.543099, -0.747668, 1.570796, 1.742589],accel_mss,speed_ms,0,blend_radius_m)
    |   movel([0.170715, -1.423477, -2.541676, -0.747236, 1.570796, 1.741512],accel_mss,speed_ms,0,blend_radius_m)
    |   movel([0.169511, -1.425278, -2.540290, -0.746821, 1.570796, 1.740307],accel_mss,speed_ms,0,blend_radius_m)
    |   movel([0.168190, -1.427015, -2.538948, -0.746426, 1.570796, 1.738986],accel_mss,speed_ms,0,blend_radius_m)
    |   movel([0.166762, -1.428684, -2.537655, -0.746050, 1.570796, 1.737559],accel_mss,speed_ms,0,blend_radius_m)
    |   movel([0.165234, -1.430277, -2.536417, -0.745696, 1.570796, 1.736030],accel_mss,speed_ms,0,blend_radius_m)
    |   movel([0.163615, -1.431789, -2.535237, -0.745363, 1.570796, 1.734411],accel_mss,speed_ms,0,blend_radius_m)
    |   movel([0.161913, -1.433215, -2.534122, -0.745052, 1.570796, 1.732709],accel_mss,speed_ms,0,blend_radius_m)
    |   movel([0.160137, -1.434547, -2.533078, -0.744764, 1.570796, 1.730933],accel_mss,speed_ms,0,blend_radius_m)
    |   movel([0.158298, -1.435778, -2.532110, -0.744501, 1.570796, 1.729094],accel_mss,speed_ms,0,blend_radius_m)
    |   movel([0.156399, -1.436906, -2.531221, -0.744262, 1.570796, 1.727195],accel_mss,speed_ms,0,blend_radius_m)
    |   movel([0.154454, -1.437924, -2.530417, -0.744047, 1.570796, 1.725250],accel_mss,speed_ms,0,blend_radius_m)
    |   movel([0.152467, -1.438824, -2.529706, -0.743859, 1.570796, 1.723263],accel_mss,speed_ms,0,blend_radius_m)
    |   movel([0.150445, -1.439600, -2.529091, -0.743698, 1.570796, 1.721242],accel_mss,speed_ms,0,blend_radius_m)
    |   movel([0.148397, -1.440248, -2.528577, -0.743564, 1.570796, 1.719194],accel_mss,speed_ms,0,blend_radius_m)
    |   movel([0.146334, -1.440759, -2.528171, -0.743459, 1.570796, 1.717131],accel_mss,speed_ms,0,blend_radius_m)
    |   # Splitting Linear movement in 28 (instruction 295: MoveL 264)
    |   movel([0.144149, -1.441227, -2.527799, -0.743363, 1.570796, 1.714945],accel_mss,speed_ms,0,blend_radius_m)
    |   movel([0.141963, -1.441698, -2.527424, -0.743267, 1.570796, 1.712760],accel_mss,speed_ms,0,blend_radius_m)
    |   movel([0.139779, -1.442173, -2.527046, -0.743170, 1.570796, 1.710575],accel_mss,speed_ms,0,blend_radius_m)
    |   movel([0.137595, -1.442651, -2.526665, -0.743073, 1.570796, 1.708391],accel_mss,speed_ms,0,blend_radius_m)
    |   movel([0.135412, -1.443132, -2.526281, -0.742976, 1.570796, 1.706208],accel_mss,speed_ms,0,blend_radius_m)
    |   movel([0.133229, -1.443617, -2.525894, -0.742878, 1.570796, 1.704025],accel_mss,speed_ms,0,blend_radius_m)
    |   movel([0.131047, -1.444106, -2.525503, -0.742780, 1.570796, 1.701843],accel_mss,speed_ms,0,blend_radius_m)
    |   movel([0.128865, -1.444597, -2.525110, -0.742682, 1.570796, 1.699662],accel_mss,speed_ms,0,blend_radius_m)
    |   movel([0.126685, -1.445092, -2.524714, -0.742583, 1.570796, 1.697481],accel_mss,speed_ms,0,blend_radius_m)
    |   movel([0.124505, -1.445591, -2.524314, -0.742484, 1.570796, 1.695301],accel_mss,speed_ms,0,blend_radius_m)
    |   movel([0.122325, -1.446092, -2.523912, -0.742385, 1.570796, 1.693122],accel_mss,speed_ms,0,blend_radius_m)
    |   movel([0.120147, -1.446597, -2.523506, -0.742286, 1.570796, 1.690943],accel_mss,speed_ms,0,blend_radius_m)
    |   movel([0.117969, -1.447105, -2.523098, -0.742186, 1.570796, 1.688765],accel_mss,speed_ms,0,blend_radius_m)
    |   movel([0.115792, -1.447617, -2.522686, -0.742086, 1.570796, 1.686588],accel_mss,speed_ms,0,blend_radius_m)
    |   movel([0.113616, -1.448131, -2.522271, -0.741986, 1.570796, 1.684412],accel_mss,speed_ms,0,blend_radius_m)
    |   movel([0.111441, -1.448649, -2.521854, -0.741886, 1.570796, 1.682237],accel_mss,speed_ms,0,blend_radius_m)
    |   movel([0.109266, -1.449171, -2.521433, -0.741785, 1.570796, 1.680063],accel_mss,speed_ms,0,blend_radius_m)
    |   movel([0.107093, -1.449695, -2.521010, -0.741684, 1.570796, 1.677889],accel_mss,speed_ms,0,blend_radius_m)
    |   movel([0.104920, -1.450223, -2.520583, -0.741583, 1.570796, 1.675716],accel_mss,speed_ms,0,blend_radius_m)
    |   movel([0.102748, -1.450754, -2.520153, -0.741482, 1.570796, 1.673545],accel_mss,speed_ms,0,blend_radius_m)
    |   movel([0.100577, -1.451288, -2.519720, -0.741381, 1.570796, 1.671374],accel_mss,speed_ms,0,blend_radius_m)
    |   movel([0.098407, -1.451825, -2.519285, -0.741280, 1.570796, 1.669204],accel_mss,speed_ms,0,blend_radius_m)
    |   movel([0.096238, -1.452365, -2.518846, -0.741178, 1.570796, 1.667035],accel_mss,speed_ms,0,blend_radius_m)
    |   movel([0.094070, -1.452908, -2.518404, -0.741076, 1.570796, 1.664867],accel_mss,speed_ms,0,blend_radius_m)
    |   movel([0.091903, -1.453455, -2.517960, -0.740974, 1.570796, 1.662700],accel_mss,speed_ms,0,blend_radius_m)
    |   movel([0.089738, -1.454005, -2.517512, -0.740872, 1.570796, 1.660534],accel_mss,speed_ms,0,blend_radius_m)
    |   movel([0.087573, -1.454557, -2.517061, -0.740770, 1.570796, 1.658369],accel_mss,speed_ms,0,blend_radius_m)
    |   movel([0.085409, -1.455113, -2.516608, -0.740668, 1.570796, 1.656205],accel_mss,speed_ms,0,blend_radius_m)
    |   movel([0.083905, -1.455522, -2.516273, -0.740593, 1.570796, 1.654702],accel_mss,speed_ms,0,blend_radius_m)
    |   movel([0.083590, -1.455504, -2.516289, -0.740596, 1.570796, 1.654387],accel_mss,speed_ms,0,blend_radius_m)
    |   movel([0.083340, -1.455371, -2.516398, -0.740621, 1.570796, 1.654136],accel_mss,speed_ms,0,blend_radius_m)
    |   movel([0.083173, -1.455091, -2.516626, -0.740672, 1.570796, 1.653970],accel_mss,speed_ms,0,blend_radius_m)
    |   movel([0.083159, -1.454077, -2.517453, -0.740859, 1.570796, 1.653955],accel_mss,speed_ms,0,blend_radius_m)
    |   movel([0.083312, -1.453634, -2.517814, -0.740941, 1.570796, 1.654109],accel_mss,speed_ms,0,blend_radius_m)
    |   movel([0.083555, -1.453287, -2.518096, -0.741005, 1.570796, 1.654351],accel_mss,speed_ms,0,blend_radius_m)
    |   movel([0.083875, -1.453020, -2.518313, -0.741055, 1.570796, 1.654671],accel_mss,speed_ms,0,blend_radius_m)
    |   movel([0.084695, -1.452650, -2.518614, -0.741124, 1.570796, 1.655492],accel_mss,speed_ms,0,blend_radius_m)
    |   movel([0.085672, -1.452382, -2.518832, -0.741175, 1.570796, 1.656468],accel_mss,speed_ms,0,blend_radius_m)
    |   # Splitting Linear movement in 26 (instruction 306: MoveL 275)
    |   movel([0.087929, -1.451800, -2.519305, -0.741284, 1.570796, 1.658725],accel_mss,speed_ms,0,blend_radius_m)
    |   movel([0.090187, -1.451222, -2.519773, -0.741393, 1.570796, 1.660983],accel_mss,speed_ms,0,blend_radius_m)
    |   movel([0.092446, -1.450647, -2.520239, -0.741502, 1.570796, 1.663242],accel_mss,speed_ms,0,blend_radius_m)
    |   movel([0.094706, -1.450076, -2.520702, -0.741611, 1.570796, 1.665502],accel_mss,speed_ms,0,blend_radius_m)
    |   movel([0.096967, -1.449508, -2.521161, -0.741720, 1.570796, 1.667764],accel_mss,speed_ms,0,blend_radius_m)
    |   movel([0.099230, -1.448943, -2.521617, -0.741829, 1.570796, 1.670026],accel_mss,speed_ms,0,blend_radius_m)
    |   movel([0.101493, -1.448382, -2.522069, -0.741937, 1.570796, 1.672290],accel_mss,speed_ms,0,blend_radius_m)
    |   movel([0.103758, -1.447824, -2.522519, -0.742046, 1.570796, 1.674554],accel_mss,speed_ms,0,blend_radius_m)
    |   movel([0.106023, -1.447270, -2.522965, -0.742154, 1.570796, 1.676819],accel_mss,speed_ms,0,blend_radius_m)
    |   movel([0.108289, -1.446719, -2.523408, -0.742262, 1.570796, 1.679086],accel_mss,speed_ms,0,blend_radius_m)
    |   movel([0.110557, -1.446172, -2.523848, -0.742369, 1.570796, 1.681353],accel_mss,speed_ms,0,blend_radius_m)
    |   movel([0.112825, -1.445628, -2.524284, -0.742477, 1.570796, 1.683621],accel_mss,speed_ms,0,blend_radius_m)
    |   movel([0.115094, -1.445088, -2.524717, -0.742584, 1.570796, 1.685891],accel_mss,speed_ms,0,blend_radius_m)
    |   movel([0.117364, -1.444551, -2.525147, -0.742691, 1.570796, 1.688161],accel_mss,speed_ms,0,blend_radius_m)
    |   movel([0.119635, -1.444018, -2.525574, -0.742798, 1.570796, 1.690432],accel_mss,speed_ms,0,blend_radius_m)
    |   movel([0.121907, -1.443488, -2.525997, -0.742904, 1.570796, 1.692704],accel_mss,speed_ms,0,blend_radius_m)
    |   movel([0.124180, -1.442962, -2.526417, -0.743010, 1.570796, 1.694976],accel_mss,speed_ms,0,blend_radius_m)
    |   movel([0.126453, -1.442439, -2.526834, -0.743116, 1.570796, 1.697250],accel_mss,speed_ms,0,blend_radius_m)
    |   movel([0.128728, -1.441920, -2.527247, -0.743221, 1.570796, 1.699524],accel_mss,speed_ms,0,blend_radius_m)
    |   movel([0.131003, -1.441405, -2.527657, -0.743327, 1.570796, 1.701799],accel_mss,speed_ms,0,blend_radius_m)
    |   movel([0.133279, -1.440894, -2.528064, -0.743431, 1.570796, 1.704075],accel_mss,speed_ms,0,blend_radius_m)
    |   movel([0.135555, -1.440386, -2.528468, -0.743536, 1.570796, 1.706351],accel_mss,speed_ms,0,blend_radius_m)
    |   movel([0.137832, -1.439881, -2.528868, -0.743640, 1.570796, 1.708629],accel_mss,speed_ms,0,blend_radius_m)
    |   movel([0.140110, -1.439381, -2.529265, -0.743744, 1.570796, 1.710906],accel_mss,speed_ms,0,blend_radius_m)
    |   movel([0.142389, -1.438884, -2.529658, -0.743847, 1.570796, 1.713185],accel_mss,speed_ms,0,blend_radius_m)
    |   movel([0.144668, -1.438390, -2.530049, -0.743950, 1.570796, 1.715464],accel_mss,speed_ms,0,blend_radius_m)
    |   movel([0.146571, -1.437942, -2.530403, -0.744044, 1.570796, 1.717367],accel_mss,speed_ms,0,blend_radius_m)
    |   movel([0.148451, -1.437412, -2.530822, -0.744155, 1.570796, 1.719247],accel_mss,speed_ms,0,blend_radius_m)
    |   movel([0.150313, -1.436788, -2.531314, -0.744287, 1.570796, 1.721109],accel_mss,speed_ms,0,blend_radius_m)
    |   movel([0.152157, -1.436061, -2.531887, -0.744441, 1.570796, 1.722953],accel_mss,speed_ms,0,blend_radius_m)
    |   movel([0.153985, -1.435217, -2.532551, -0.744621, 1.570796, 1.724781],accel_mss,speed_ms,0,blend_radius_m)
    |   movel([0.155798, -1.434249, -2.533312, -0.744829, 1.570796, 1.726594],accel_mss,speed_ms,0,blend_radius_m)
    |   movel([0.157601, -1.433140, -2.534180, -0.745068, 1.570796, 1.728398],accel_mss,speed_ms,0,blend_radius_m)
    |   movel([0.159392, -1.431885, -2.535162, -0.745342, 1.570796, 1.730189],accel_mss,speed_ms,0,blend_radius_m)
    |   movel([0.161799, -1.429920, -2.536694, -0.745775, 1.570796, 1.732595],accel_mss,speed_ms,0,blend_radius_m)
    |   movel([0.163946, -1.427834, -2.538314, -0.746241, 1.570796, 1.734742],accel_mss,speed_ms,0,blend_radius_m)
    |   movel([0.165825, -1.425650, -2.540003, -0.746736, 1.570796, 1.736622],accel_mss,speed_ms,0,blend_radius_m)
    |   movel([0.167436, -1.423394, -2.541740, -0.747255, 1.570796, 1.738232],accel_mss,speed_ms,0,blend_radius_m)
    |   movel([0.168771, -1.421092, -2.543505, -0.747792, 1.570796, 1.739568],accel_mss,speed_ms,0,blend_radius_m)
    |   movel([0.169823, -1.418777, -2.545271, -0.748341, 1.570796, 1.740619],accel_mss,speed_ms,0,blend_radius_m)
    |   movel([0.170587, -1.416471, -2.547023, -0.748895, 1.570796, 1.741383],accel_mss,speed_ms,0,blend_radius_m)
    |   movel([0.171055, -1.414208, -2.548735, -0.749447, 1.570796, 1.741851],accel_mss,speed_ms,0,blend_radius_m)
    |   movel([0.171221, -1.412013, -2.550387, -0.749989, 1.570796, 1.742017],accel_mss,speed_ms,0,blend_radius_m)
    |   movel([0.171077, -1.409918, -2.551957, -0.750513, 1.570796, 1.741873],accel_mss,speed_ms,0,blend_radius_m)
    |   movel([0.170618, -1.407957, -2.553422, -0.751010, 1.570796, 1.741414],accel_mss,speed_ms,0,blend_radius_m)
    |   movel([0.169835, -1.406156, -2.554762, -0.751471, 1.570796, 1.740631],accel_mss,speed_ms,0,blend_radius_m)
    |   movel([0.168721, -1.404552, -2.555951, -0.751886, 1.570796, 1.739517],accel_mss,speed_ms,0,blend_radius_m)
    |   movel([0.167272, -1.403171, -2.556972, -0.752246, 1.570796, 1.738068],accel_mss,speed_ms,0,blend_radius_m)
    |   movel([0.165480, -1.402051, -2.557798, -0.752540, 1.570796, 1.736276],accel_mss,speed_ms,0,blend_radius_m)
    |   movel([0.163342, -1.401219, -2.558410, -0.752760, 1.570796, 1.734139],accel_mss,speed_ms,0,blend_radius_m)
    |   # Splitting Linear movement in 6 (instruction 331: MoveL 300)
    |   movel([0.161964, -1.400830, -2.558696, -0.752863, 1.570796, 1.732760],accel_mss,speed_ms,0,blend_radius_m)
